# B&R Automation Studio project EFI (part 16)

#### pressureControl.st - Pressure control PID
```iecst
ACTION pressureControl:

	IF inks.parameters.StartUp.xActive THEN
		rMeniscusSp := inks._Internal.Startup.rSetPointMeniscus;
	ELSE
		rMeniscusSp := inks.parSw.NegPump.rSetPointMeniscus;
	END_IF

	xReservoirParamsNeeded := xPressureReservoirStable OR (xReservoirModeActivated AND  mode9); //INKS_STOPPING

	parPidMeniscus:=stPIDParamId(parBar.paramsPidMeniscus);
	xUpdatePidMeniscus:= parPidMeniscusCopy <> parPidMeniscus;
	parPidMeniscusCopy:=parPidMeniscus;
	IF xUpdatePidMeniscus THEN
		iQuantityUpdatePidMeniscus:=iQuantityUpdatePidMeniscus+1;
	END_IF;
	IF xUpdatePidMeniscus OR EDGE(xReservoirParamsNeeded) THEN
		IF NOT xReservoirParamsNeeded THEN
			//Standart values
			stPIDParamToMTPIDParameters(ADR(parBar.paramsPidMeniscus), ADR(pidParMeniscus));
		ELSE
			stPIDParamToMTPIDParameters(ADR(parBar.paramsPidMeniscusReservoir), ADR(pidParMeniscus));
		END_IF
	END_IF;

	parPidPos:=stPIDParamId(parBar.paramsPidPositive);
	xUpdatePidPos:= parPidPosCopy <> parPidPos;
	parPidPosCopy:=parPidPos;
	IF xUpdatePidPos THEN
		iQuantityUpdatePidPos:=iQuantityUpdatePidPos+1;
	END_IF;
	IF xUpdatePidPos OR EDGE(xReservoirParamsNeeded) THEN
		IF NOT xReservoirParamsNeeded THEN
			//Standart values
			stPIDParamToMTPIDParameters(ADR(parBar.paramsPidPositive), ADR(pidParPresPos));
		ELSE
			stPIDParamToMTPIDParameters(ADR(parBar.paramsPidPositiveReservoir), ADR(pidParPresPos));
		END_IF
	END_IF;

	TON_ExecutionDelay(IN:=TRUE, PT:= T#100MS);

	//timer to change the management of the filling pump.
	//Issue 1813: Modification in the change filling control condition, now if the difference between Sp and real meniscus is equal to zero, we change to PID control, too.
	//
	TON_ChangeFillingControl(	IN:=( mode3 AND NOT inks.parameters.Priming.xSystemNeedsPriming AND (rMeniscusError <  LC_MAX_MENISCUS_TO_STARTED)) AND
									( mode3 AND NOT inks.parameters.Priming.xSystemNeedsPriming AND (rMeniscusError >= LC_MIN_MENISCUS_TO_STARTED)) ,
								PT:= T#0.1S);
	IF NOT mode3 THEN
		xGoToStarted := FALSE;
	ELSIF TON_ChangeFillingControl.Q THEN
		xGoToStarted := TRUE;
	END_IF

	IF mode3 AND NOT xPrimingStabilized AND
		( inks.status.PosPump.rDutyCycleFilling > inks.parameters.PosPump.rDCThresholdPriming) AND
		( (rSPfillingPump <> rSP_PressurePos_PID) OR (rMeniscusSp <> rSP_Meniscus_PID) ) THEN

		xPrimingStabilized:=TRUE;
	END_IF

	//Modify the Positive SetPoint during starting
	pressPosAcceleration;

	//**********************************************************************************
	//It changes SP maniscus when is detected differential pressure lower than 20mbars
	//**********************************************************************************
	IF NOT xDrippingOrder THEN

		IF inks.parameters.Priming.xSystemNeedsPriming THEN

			IF mode4 THEN //Inks Started

				// Timer management	for controlling changes in meniscus SP
				TON_ChangeSPstarting(IN:= ( xPrimingStabilized AND (NOT TON_ChangeSPstarting.Q) ), PT:= T#300MS);
				xUpdateSpPriming:= TON_ChangeSPstarting.Q AND inks.status.Temp.rTemp > (rSPtemp-4);

				rPressurePos:= ABS (inks.status.rVacuum1-rSP_PressurePos_PID);
				IF xUpdateSpPriming AND ( rPressurePos < inks.parameters.Priming.rThresholdPressure ) AND (rSPfillingPump <> rSP_PressurePos_PID)  THEN
					// rSPfillingPump is POS PRESSURE SP from GUI

					// rSP_PressurePos_PID current positive pressure sensor
					IF (rSPfillingPump < rSP_PressurePos_PID) THEN
						//Decrease Pos and Meniscus SPs
						rSP_PosPrimStabilizing := rSP_PosPrimStabilizing - 1;
					ELSE
						//Decrease Pos and Meniscus SPs
						rSP_PosPrimStabilizing := rSP_PosPrimStabilizing + 1;
					END_IF
				END_IF

				rPressureMen:= ABS (inks.status.rMeniscus-rSP_Meniscus_PID);
				IF xUpdateSpPriming AND ( rPressureMen < inks.parameters.Priming.rThresholdPressure ) AND  (rMeniscusSp <> rSP_Meniscus_PID) AND (rSPfillingPump = rSP_PressurePos_PID) THEN

					IF (rMeniscusSp < rSP_Meniscus_PID) THEN
						//Decrease Pos and Meniscus SPs
						rSP_NegPrimStabilizing := rSP_NegPrimStabilizing - 1;
					ELSE
						//Decrease Pos and Meniscus SPs
						rSP_NegPrimStabilizing := rSP_NegPrimStabilizing + 1;
					END_IF
				END_IF

				//Update de SetPoints of the PID
				rSP_Meniscus_PID:=rSP_NegPrimStabilizing;
				rSP_PressurePos_PID:=rSP_PosPrimStabilizing;

			END_IF

		ELSE	// THIS IS THE CASE WITHOUT THE PRIMING, THE STANDART BEHAVIOR

			IF xStateReverseFlow THEN

				IF (inks.status.rDeltaPressure <= 20.0) THEN
					rSP_PressurePos_PID := -15.0;
					rSP_Meniscus_PID := 25.0;
				ELSE
					inks.status.startChangeSPInDelta:=TRUE;
				END_IF

			ELSE
				rSP_PressurePos_PID:= rSPfillingPump;
				rSP_Meniscus_PID:=rMeniscusSp;
			END_IF

			// Timer management
			TON_ChangeSPInDelta(IN:=inks.status.startChangeSPInDelta, PT:= SECONDS_TO_TIME(inks.parameters.iTimeChangeSPInRev));
			IF TON_ChangeSPInDelta.Q THEN
				rSP_PressurePos_PID:= rSPfillingPump;
				rSP_Meniscus_PID:=rMeniscusSp;
				inks.status.startChangeSPInDelta:=FALSE;
			END_IF

		END_IF

	ELSE //The ink System has DRIP ORDER

		rSP_Meniscus_PID:=SETPOINT_MENISCUS_DRIP;
		rSP_PressurePos_PID:= -SETPOINT_MENISCUS_DRIP + rSPfillingPump + rMeniscusSp;
		xPrimingStabilized:=FALSE;

	END_IF

	//VACUUM - NEGATIVE - VACUUM - NEGATIVE - VACUUM - NEGATIVE - VACUUM - NEGATIVE - VACUUM - NEGATIVE -
	//VACUUM - NEGATIVE - VACUUM - NEGATIVE - VACUUM - NEGATIVE - VACUUM - NEGATIVE - VACUUM - NEGATIVE -

	//negative pump management.
	iReasonEnableNegPID.0 := mode3;
	iReasonEnableNegPID.1 := mode4;
	iReasonEnableNegPID.2 := mode5;
	iReasonEnableNegPID.3 := mode6;
	iReasonEnableNegPID.4 := mode9;
	xEnableNegPID := iReasonEnableNegPID > 0;

	xHoldMeniscus := (inks.status.iDirection = INKSDIR_REVERSE AND NOT TON_StabSolPid1Neg.Q) OR
					(	NOT TON_StabSolPid2Neg.Q AND
					mode4 AND //INKS_STARTED
					xStateReverseFlow);

	//**********************************************************************************
	// PID PID PID PID PID PID PID PID PID PID PID PID PID PID PID PID PID PID PID PID
	//**********************************************************************************
	fb_PID_Pres(Enable:=xEnableNegPID AND TON_ExecutionDelay.Q,
						PIDParameters:=pidParMeniscus,
						HoldOut:= xHoldMeniscus,
						MinOut:=0.0,
						MaxOut:=100.0,
						Update:= xUpdatePidMeniscus,
						SetValue:=rSP_Meniscus_PID,
						ActValue:=rMeniscusPV
						);
	rOrderBNegative:=fb_PID_Pres.Out;

	//POSITIVE - POSITIVE - POSITIVE - POSITIVE - POSITIVE - POSITIVE - POSITIVE - POSITIVE - POSITIVE - POSITIVE -
	//POSITIVE - POSITIVE - POSITIVE - POSITIVE - POSITIVE - POSITIVE - POSITIVE - POSITIVE - POSITIVE - POSITIVE -

	//filling pump management.
	iReasonEnablePosPID.0 := mode3 AND inks.parameters.Priming.xSystemNeedsPriming;
	iReasonEnablePosPID.1 := mode4;
	iReasonEnablePosPID.2 := mode5;
	iReasonEnablePosPID.3 := mode6;
	iReasonEnablePosPID.4 := mode9;
	xEnablePosPID := iReasonEnablePosPID > 0;

	xHoldPos:= (inks.status.iDirection = INKSDIR_REVERSE AND NOT TON_StabSolPid1Pos.Q) OR
				(NOT TON_StabSolPid2Pos.Q AND
				mode4 AND //INKS_STARTED
				xStateReverseFlow	);

	//**********************************************************************************
	// PID PID PID PID PID PID PID PID PID PID PID PID PID PID PID PID PID PID PID PID
	//**********************************************************************************
	fb_PID_PresFilling(Enable:=xEnablePosPID AND TON_ExecutionDelay.Q,
						PIDParameters:=pidParPresPos,
						HoldOut:= xHoldPos,
						MinOut:=0.0,
						MaxOut:=100.0,
						Update:= xUpdatePidPos,
						SetValue:=rSP_PressurePos_PID,
						ActValue:=rPressureCollectorPos1
						);
	rOrderBPositive:=fb_PID_PresFilling.Out;

	//Define the pump outputs depending on the state

	IF mode3 THEN
		IF inks.parameters.Priming.xSystemNeedsPriming THEN
			rSP_Meniscus_PID	:= inks.parameters.NegPump.rSetPointPrimingStarting;
			rSP_PressurePos_PID	:= inks.parameters.PosPump.rSetPointPrimingStarting;
			inks.status.PosPump.rDutyCycleFilling:=rOrderBPositive;

			//Prepare the initial value for Stabilization stage
			rSP_PosPrimStabilizing:=inks.parameters.PosPump.rSetPointPrimingStarting;
			rSP_NegPrimStabilizing:=inks.parameters.NegPump.rSetPointPrimingStarting;
		ELSE
			rSetPointFillingPump:=parBar.rSPfillingPumpStarting;
			inks.status.PosPump.rDutyCycleFilling:=rOrderBPositiveStart;
		END_IF
		inks.status.NegPump.rDutyCycleNegative:=rOrderBNegative;
	END_IF

	IF NOT mode10 AND (mode4 OR mode5 OR mode6) THEN
		inks.status.PosPump.rDutyCycleFilling:=rOrderBPositive;
		inks.status.NegPump.rDutyCycleNegative:=rOrderBNegative;
	END_IF

	IF mode13 THEN
		inks.status.NegPump.rDutyCycleNegative:=inks.parameters.NegPump.rDCPriming;
		inks.status.PosPump.rDutyCycleFilling:=inks.parameters.PosPump.rDCPriming;
	END_IF

	IF mode10 THEN //InksManifoldCleaning
		inks.status.PosPump.rDutyCycleFilling:=inks.parSw.PosPump.rSetPointManual;
		inks.status.NegPump.rDutyCycleNegative:=inks.parSw.NegPump.rSetPointManual;
	END_IF

	//Sanity checks
	IF mode1 THEN //Inks Stopped
		inks.status.PosPump.rDutyCycleFilling:=0;
		inks.status.NegPump.rDutyCycleNegative:=0;
		xPrimingStabilized:=FALSE;
	END_IF

END_ACTION
```

#### conversionsPost.st - Posconversions
```iecst
ACTION conversionsPost:

	IF  inks.status.xInksRunning THEN

		//Negative Pump
		IF inks.status.NegPump.rDutyCycleNegative=0.0 THEN
			inks.signals.out.iDutyCycleNegative:=0;
		ELSE
			rVoltageNegPump:= (inks.status.NegPump.rDutyCycleNegative * rSlopePumpNeg) + rLowPumpLimitNeg;
			inks.signals.out.iDutyCycleNegative:=REAL_TO_INT(rVoltageNegPump * 32766 / 10); //10V correspond to 32766
		END_IF;

		//Positive Pump
		IF inks.status.PosPump.rDutyCycleFilling=0.0 THEN
			inks.signals.out.iDutyCycleFilling:=0;
		ELSE
			rVoltagePosPump:= (inks.status.PosPump.rDutyCycleFilling * rSlopePumpPos) + rLowPumpLimitPos;
			inks.signals.out.iDutyCycleFilling:=REAL_TO_INT(rVoltagePosPump * 32766 / 10); //10V correspond to 32766
		END_IF;

	ELSE
		inks.signals.out.iDutyCycleNegative:=0;
		inks.signals.out.iDutyCycleFilling:=0;

	END_IF;

	///vars to show in GUI
	inks.status.Tank.iDipositLevel:=REAL_TO_INT(rTankLevelPercent);
	inks.status.tiDriptime:=inks.parSw.tiDripTime;
	inks.status.PosPump.rSetPointPos:=rSP_PressurePos_PID;

	// Duty cycle Heater Tank in Percentage
	inks.status.Temp.rDutyCycleTempPowerRedTank:= inks.status.Temp.rDutyCycleTempTank;   //TOREVIEW: It doesn't seems to be OK (JMH)

END_ACTION
```

#### alarms.st - Alarms
```iecst
ACTION alarms:
	//Ink level alarm
	inks.Al.xAlrTankDigitalSensorsError := NOT inks.status.xActTestMode AND NOT inks.status.Tank.xMinLevel AND inks.status.Tank.xMaxLevel;

	//Temperature and Vacuum probe alarms
	TON_Reset(IN:= NOT xIAmInReverse AND inks.status.xInksRunning, PT:= T#1S);
	t_reset := TON_Reset.Q;

	//Silvia: added an equal symbol in the comparison, because it's impossible to have more than 150mbar.
	TON_AlrVacuum1.IN	:=	t_reset AND (rPressureCollectorPos1 >= rVacuumSensorMax) AND (inks.signals.out.iDutyCycleNegative<>0);
	TON_AlrVacuum1.PT	:=	T#1S; //T#2S; //SUSTPLATF-266
	TON_AlrVacuum1();

	IF TON_AlrVacuum1.Q THEN
		inks.Al.xAlrVacuum1 := TRUE;
	END_IF

	TON_AlrVacuum2.IN	:=	t_reset AND (rPressureCollectorPos2 >= rVacuumSensorMax) AND (inks.signals.out.iDutyCycleFilling<>0);
	TON_AlrVacuum2.PT	:=	T#1S; //T#2S; //SUSTPLATF-266
	TON_AlrVacuum2();

	IF TON_AlrVacuum2.Q THEN
		inks.Al.xAlrVacuum2 := TRUE;
	END_IF

	// Alarm Error in Vacuum gauge means that analog input status is lower than -8000
	TON_DelayVacuum1Gauge.IN	:=	inks.signals.in.xVacuum1SensorError;
	TON_DelayVacuum1Gauge.PT	:=	T#2S;
	TON_DelayVacuum1Gauge();

	IF TON_DelayVacuum1Gauge.Q THEN
		inks.Al.xAlrVacuumSensor1 := TRUE;
	END_IF

	// Alarm Error in Vacuum gauge means that analog input status is lower than -8000
	TON_DelayVacuum2Gauge.IN	:=	inks.signals.in.xVacuum2SensorError;
	TON_DelayVacuum2Gauge.PT	:=	T#2S;
	TON_DelayVacuum2Gauge();

	IF TON_DelayVacuum2Gauge.Q THEN
		inks.Al.xAlrVacuumSensor2 := TRUE;
	END_IF

	TON_AlrVacuumDiff(IN:=t_reset AND ABS(inks.status.rMeniscus-rMeniscusSp) > inks.parSw.NegPump.rLimitMeniscusDiffWarning AND
					NOT inks.Al.xAlrVacuum1 AND	NOT inks.Al.xAlrVacuum2 AND	NOT inks.commands.xErrorRst,
					PT:= T#1S);

	TON_AlrVacuumDiff2(	IN:=mode4 AND ABS(inks.status.rMeniscus-rMeniscusSp) < inks.parSw.NegPump.rLimitMeniscusDiffWarning,
						PT:= T#5S);

	IF TON_AlrVacuumDiff2.Q OR NOT inks.status.xInksRunning THEN
		inks.Al.xAlrDiffVacuum := FALSE;
	// xOrderOnReverseCapped when is cleaning while 50 secs, from start reverse to be finished
	ELSIF TON_AlrVacuumDiff.Q AND NOT xIgnoreAlarmsInCleaning AND NOT inks.status.Reverse.xOnReverseAuto THEN
		inks.Al.xAlrDiffVacuum := TRUE;
	END_IF

	//Temperature alarms management

	//Alarm in the Manifold temperature gauge. (Out of range)
	TON_AlrIncoherTempHeat.IN	:=	t_reset AND ( inks.status.Temp.rTemp < 0.0 OR inks.status.Temp.rTemp > 100.0 );
	TON_AlrIncoherTempHeat.PT	:=	T#2S;
	TON_AlrIncoherTempHeat();

	IF TON_AlrIncoherTempHeat.Q THEN
		inks.Al.xAlrIncoherTempHeat := TRUE;
	END_IF

	//Alarm in Bar Heater temperature gauge. (Out of range)
	TON_AlrTempHeaterMax.IN	:=	(inks.status.Temp.rTemp > 80.0);
	TON_AlrTempHeaterMax.PT	:=	T#2S;
	TON_AlrTempHeaterMax();

	IF TON_AlrTempHeaterMax.Q THEN
		inks.Al.xAlrHeaterReachsMaxTemp := TRUE;
	END_IF

	//////////////////////////////////////////////////////////////////////////////////////////////////////////////////////
	//Alarm of temperature gauge broken temperature gauge in collector. Error detected by the plc
	// COLLECTOR
	// Alarm Error in Vacuum gauge means that analog input status is lower than -8000
	//////////////////////////////////////////////////////////////////////////////////////////////////////////////////////
	TON_AlrTempGauge.IN	:=	(inks.signals.in.xTempSensorError);
	TON_AlrTempGauge.PT	:=	T#2S;
	TON_AlrTempGauge();

	IF TON_AlrTempGauge.Q THEN
		inks.Al.xAlrTempSensor := TRUE;
	END_IF

	alarmsTankHeater;

	//////////////////////////////////////////////////////////////////////////////////////////////////////////////////////
	// Alarm differential temperature
	//////////////////////////////////////////////////////////////////////////////////////////////////////////////////////

	//WARNING

	TON_AlrDifTemp.IN := ABS(inks.status.Temp.rTemp - rSPtemp) > MAX_DIFFCTRLTEMP_WRNG;
	TON_AlrDifTemp.PT := T#2S;
	TON_AlrDifTemp();

	TON_AlrNotDifTemp.IN :=	ABS(inks.status.Temp.rTemp-rSPtemp) < MAX_DIFFCTRLTEMP_WRNG;
	TON_AlrNotDifTemp.PT :=	T#5S;
	TON_AlrNotDifTemp();

	IF NOT inks.status.xInksRunning OR TON_AlrNotDifTemp.Q THEN
		inks.Al.xAlrDiffInCtrlTemp := FALSE;
	ELSIF TON_AlrDifTemp.Q THEN
		inks.Al.xAlrDiffInCtrlTemp := TRUE;
	END_IF

	//ALARM

	IF NOT inks.status.xInksRunning OR NOT inks.status.xEnabledBarToPrint OR TON_AlrNotDifTempExcessiv.Q THEN
		inks.Al.xAlrDifCtrlTempExcessive := FALSE;
	ELSIF TON_AlrDifTempExcessiv.Q THEN
		inks.Al.xAlrDifCtrlTempExcessive := TRUE;
	END_IF

	TON_AlrDifTempExcessiv.IN := ABS(inks.status.Temp.rTemp - rSPtemp) > MAX_DIFFCTRLTEMPHIGH_ALR;
	TON_AlrDifTempExcessiv.PT := T#20s;
	TON_AlrDifTempExcessiv();

	TON_AlrNotDifTempExcessiv.IN := ABS(inks.status.Temp.rTemp - rSPtemp) < MAX_DIFFCTRLTEMPHIGH_ALR;
	TON_AlrNotDifTempExcessiv.PT := T#20s;
	TON_AlrNotDifTempExcessiv();

	//////////////////////////////////////////////////////////////////////////////////////////////////////////////////////
	// Alarm PLC not heating bar
	//////////////////////////////////////////////////////////////////////////////////////////////////////////////////////
	tonAlrNotHeating.IN := inks.status.xInksRunning AND NOT mode10 AND
						(rSPtemp - inks.status.Temp.rTemp > MAX_DIFFCTRLTEMP_ALR) AND
						NOT inks.signals.out.xOutBarResistance;
	tonAlrNotHeating.PT := T#1m;
	tonAlrNotHeating();
	IF tonAlrNotHeating.Q THEN
		IF NOT inks.Al.xAlrHeaterOutFault THEN
			//Added into the IF to avoid a double register while stopping
			LogNotHeating;
		END_IF
		inks.Al.xAlrHeaterOutFault := TRUE;
	END_IF

	//////////////////////////////////////////////////////////////////////////////////////////////////////////////////////
	//Overpressure alarm management
	//////////////////////////////////////////////////////////////////////////////////////////////////////////////////////
	TON_OverPressureDelay.IN := NOT mode1 AND inks.signals.in.xOverpressure;
	TON_OverPressureDelay.PT := T#100ms;
	TON_OverPressureDelay();

	IF TON_OverPressureDelay.Q THEN
		inks.Al.xAlrOverPressure := TRUE;
	END_IF

	//////////////////////////////////////////////////////////////////////////////////////////////////////////////////////
	//Stop Recirculation because there is not ink inn tank
	//////////////////////////////////////////////////////////////////////////////////////////////////////////////////////
	IF (mode3 OR mode13 OR mode4) AND NOT inks.status.Tank.xMinLevel AND NOT inks.status.xActTestMode THEN
		inks.Al.xAlrStopRecircNoInk:=TRUE;
	ELSIF inks.status.Tank.xMinLevel THEN
		inks.Al.xAlrStopRecircNoInk:=FALSE;
	END_IF

	//////////////////////////////////////////////////////////////////////////////////////////////////////////////////////
	// It is defined in controlMode.str_start_inks(CLK:= inks.ordersSw.xStartInks);
	// RECIRCULATION CANNOT START, INK TANK EMPTY
	//////////////////////////////////////////////////////////////////////////////////////////////////////////////////////
	IF NOT inks.status.xActTestMode AND NOT inks.status.Tank.xMinLevel AND r_start_inks.Q THEN
		inks.Al.xAlrInksRunnig:=TRUE; //To review with Jorge, this alarm is not shared in VarsVersion but exists in PLC2Kernel
	END_IF

	//////////////////////////////////////////////////////////////////////////////////////////////////////////////////////
	// Implemented 09/19/2017
	// Here, an alarm No Recirculation in the Bar is reported when is Ink system is stopped with bar installed
	// RECIRCULATION STOPPED / UNSTABLE INK SYSTEM
		//////////////////////////////////////////////////////////////////////////////////////////////////////////////////////
	inks.Al.xAlrNoRecirculation :=  NOT inks.status.xInksRunning;

	//////////////////////////////////////////////////////////////////////////////////////////////////////////////////////
	//INK SYSTEM STOPED WITH BAR ENABLE TO PRINT
	//////////////////////////////////////////////////////////////////////////////////////////////////////////////////////
	IF NOT inks.status.xInksRunning AND inks.status.xEnabledBarToPrint THEN
		inks.Al.xAlrNoRecircStop := TRUE;
	END_IF

	//////////////////////////////////////////////////////////////////////////////////////////////////////////////////////
	//Alarm to indicate that we don't allow to enter in the  manifold cleaning mode if there is no ink.
		//////////////////////////////////////////////////////////////////////////////////////////////////////////////////////
	IF NOT inks.status.xActTestMode AND NOT inks.status.Tank.xMinLevel AND EDGEPOS(inks.ordersSw.xStartManual) THEN
		inks.Al.xAlrNoInkNoCleanManif := TRUE;
	END_IF

	// rSPfillingPump is POS PRESSURE SP from GUI
	// rSP_PressurePos_PID current positive pressure sensor
	// rMeniscusSp is Meniscus SP from GUI
	// rSP_Meniscus_PID current meniscus pressure
	xOutOfCriticalRange := 	mode4 AND (rSPfillingPump = rSP_PressurePos_PID) AND (rMeniscusSp = rSP_Meniscus_PID) AND
				( rMeniscusPV > inks.parSw.NegPump.rUpperLimMeniscusCritical  OR  rMeniscusPV < inks.parSw.NegPump.rLowerLimMeniscusCritical );

	TON_AlrCriticalMeniscus2.IN:=t_reset AND mode4 AND NOT xIgnoreAlarmsInCleaning AND xOutOfCriticalRange;
	TON_AlrCriticalMeniscus2.PT:=T#5S;
	TON_AlrCriticalMeniscus2();

	IF TON_AlrCriticalMeniscus2.Q THEN
		inks.Al.xAlrBrokenMeniscus := TRUE;
	END_IF

	IF inks.status.xActTestMode THEN
		inks.Al.xAlrLevelSensorError := FALSE;
	ELSIF inks.status.Tank.xMaxLevel AND NOT inks.status.Tank.xMinLevel THEN
		inks.Al.xAlrLevelSensorError := TRUE;
	END_IF

	// It is not a stop alarm just warning
	inks.Al.xAlrTankToFillIn := NOT inks.status.xActTestMode AND NOT inks.status.Tank.xMaxLevel;

	// It has been improved to avoid zero state in the machine when this alarm is activated. Added condition status is different to mode1
	// 22-10-1017: Changed for commissioning SN1 at Marco Polo: It is alarm stop when inkState is different to INKS_STOPPED
	inks.Al.xAlrTankEmpty := NOT inks.status.xActTestMode AND NOT mode1 AND NOT inks.status.Tank.xMinLevel;

	// The ink level is close to Empty. Raising an alarm to allow the Machine or the line to stop production without stopping the inkSystem
	inks.Al.xAlrTankCloseToEmpty := NOT inks.status.xActTestMode AND NOT mode1 AND NOT inks.status.Tank.xCloseToMinLevel;

	TON_TimeAlrDCStarting(IN:=mode3, PT:= T#60S);  //After start, delay 60seconds taking care of this alarm

	xModesAlrDC:=TON_TimeAlrDCStarting.Q OR (mode4 AND NOT xIgnoreAlarmsInCleaning );

	TON_AlrDCDiff.IN:= xModesAlrDC AND ABS(inks.status.PosPump.rDutyCycleFilling - inks.status.NegPump.rDutyCycleNegative) > lc_rDiffBetweenPumpsDCLimit;
	TON_AlrDCDiff.PT:= inks.parameters.parBar.iTimeToActiveDcErrorAlarm;
	TON_AlrDCDiff();

	TON_AlrNegDiff.IN:= xModesAlrDC AND ( (inks.status.NegPump.rDutyCycleNegative>99) OR (inks.status.NegPump.rDutyCycleNegative < 1 ));
	TON_AlrNegDiff.PT:= inks.parameters.parBar.iTimeToActiveDcErrorAlarm;
	TON_AlrNegDiff();

	TON_AlrPosDiff.IN:= xModesAlrDC AND ( (inks.status.PosPump.rDutyCycleFilling>99) OR (inks.status.PosPump.rDutyCycleFilling < 1 ));
	TON_AlrPosDiff.PT:= inks.parameters.parBar.iTimeToActiveDcErrorAlarm;
	TON_AlrPosDiff();

	IF TON_AlrDCDiff.Q OR TON_AlrNegDiff.Q OR TON_AlrPosDiff.Q THEN
		inks.Al.xAlrPumpsDCError := TRUE;
		LogPumpDCError; //Logging the source of the Pump DC Error
	END_IF

	IF inks.signals.in.xKlixonTriggered THEN
		inks.Al.xAlrKlixonTriggered:=TRUE;
	// This ELSE must be reviewed with Dani Moya, added during Cube start up.
	ELSE
		inks.Al.xAlrKlixonTriggered:=FALSE;
	END_IF

	// It allows detection because PsuOk is delayed when is in failure
	TON_StabPsuOk.IN:=(inks.ordersSw.xPowPrintHead AND inks.signals.out.xOutPowPrintHead AND NOT inks.signals.in.xPrintHeadsPsuOK);
	TON_StabPsuOk.PT:=lc_tiTimeStoppingPsu;
	TON_StabPsuOk();

	IF TON_StabPsuOk.Q THEN
		inks.Al.xAlrPrintHeadPsuFailure:=TRUE;
	END_IF

	//DELOREAN-1961: Warning when bar enabled to print and maintenance mode active
	IF inks.status.xActMaintenanceMode AND inks.status.xEnabledBarToPrint THEN
		inks.Al.xAlrMaintenanceModeActive := TRUE;
	END_IF

	// NOZOMITWO-1410 Chiller alarms
	TON_AlrHeaterOFF.IN := inks.status.xInksRunning AND inks.parameters.InksChiller.Status=CHILLER_RUNNING AND inks.signals.out.xHeatingActive AND inks.status.Temp.rDutyCycleTemp = 0 AND (inks.parSw.Temp.rSetPointTemp + 1) < inks.status.Temp.rTemp;
	TON_AlrHeaterOFF.PT := T#120s;
	TON_AlrHeaterOFF();

	inks.Al.xHeaterOff := TON_AlrHeaterOFF.Q;

	// NOZOMITWO-1410 Chiller warnings and NOZOMITWO-2353
	TON_AlrChillerPrintheadsOFF.IN := inks.parameters.PrintheadsChiller.iIndex > 0 AND
									inks.parameters.PrintheadsChiller.Status <> CHILLER_RUNNING AND
									inks.parameters.PrintheadsChiller.Status <> CHILLER_STOPPING AND
									inks.signals.out.xOutPowPrintHead;
	TON_AlrChillerPrintheadsOFF.PT := T#30s;
	TON_AlrChillerPrintheadsOFF();

	IF TON_AlrChillerPrintheadsOFF.Q THEN
		inks.Al.xAlrPrintHeadsChillerStopped := TRUE;
	END_IF

END_ACTION

ACTION alarmsTankHeater:

	IF NOT inks.parSw.Temp.xTankHeaterEnabled THEN
		inks.Al.xAlrTempTankSensor			:= FALSE;
		inks.Al.xAlrHeaterTankReachsMaxTemp	:= FALSE;
		inks.Al.xAlrDiffInCtrlTempTank		:= FALSE;
		inks.Al.xAlrIncoherTempTank			:= FALSE;
		RETURN;
	END_IF

	//////////////////////////////////////////////////////////////////////////////////////////////////////////////////////
	//Alarm temperature gauge broken in heater or temperature gauge broken HEATER TANK. Error detected by the plc.
	// xTempTankSensorError --> It has not I/O mapping. Pending to define in P4	by EEteam
	//HEATER TANK
	//////////////////////////////////////////////////////////////////////////////////////////////////////////////////////

	TON_AlrTempTankTempSensorError.IN	:=	inks.signals.in.xTempTankSensorError;
	TON_AlrTempTankTempSensorError.PT	:=	T#2S;
	TON_AlrTempTankTempSensorError();

	// If not installed bar en It is not an alarm
	IF TON_AlrTempTankTempSensorError.Q THEN
		inks.Al.xAlrTempTankSensor := TRUE;
	END_IF

	//Alarm in Heater Tank temperature gauge. (Out of range)
	TON_AlrTempTankMax.IN	:=	(inks.status.Temp.rTempTank > 70.0);
	TON_AlrTempTankMax.PT	:=	T#2S;
	TON_AlrTempTankMax();

	IF TON_AlrTempTankMax.Q THEN
		inks.Al.xAlrHeaterTankReachsMaxTemp := TRUE;
	END_IF

	//Alarm differential temperature in tank
	TON_AlrDifTempTank.IN	:=	t_reset AND ( ABS(inks.status.Temp.rTempTank - rSPTempTank) > MAX_DIFFCTRLTEMP_WRNG);
	TON_AlrDifTempTank.PT	:=	T#2S;
	TON_AlrDifTempTank();

	TON_AlrDifTempTank2.IN	:=	inks.status.xInksRunning AND (ABS(inks.status.Temp.rTempTank-rSPTempTank) < MAX_DIFFCTRLTEMP_WRNG);
	TON_AlrDifTempTank2.PT	:=	T#5S;
	TON_AlrDifTempTank2();

	IF NOT inks.status.xInksRunning OR TON_AlrDifTempTank2.Q THEN
		inks.Al.xAlrDiffInCtrlTempTank := FALSE;
	ELSIF TON_AlrDifTempTank.Q THEN
		inks.Al.xAlrDiffInCtrlTempTank := TRUE;
	END_IF

	//Alarm in the heater tank temperature gauge. (Out of range)
	TON_AlrIncoherTempTank.IN	:=	t_reset AND ( inks.status.Temp.rTempTank < 0.0 OR inks.status.Temp.rTempTank > 100.0 );
	TON_AlrIncoherTempTank.PT	:=	T#2S;
	TON_AlrIncoherTempTank();

	IF TON_AlrIncoherTempTank.Q THEN
		inks.Al.xAlrIncoherTempTank := TRUE;
	END_IF
END_ACTION

ACTION LogPumpDCError:

	IF inks.status.NegPump.rDutyCycleNegative>99 THEN
		stEventLogNeg.Source := ELOG_TYPE_BAR;
		stEventLogNeg.Severity:= ELOG_SEVERITY_ERROR;
		stEventLogNeg.Facility:= gIndexInks;
		stEventLogNeg.ErrorCode:=0;
		stEventLogNeg.Text := 'Negative Pump in Max Value. Bar ';
		brsftoa(gIndexInks, ADR(strAux));
		brsstrcat(ADR(stEventLogNeg.Text), ADR(strAux));
		gEventLogLoader(EventData := ADR(stEventLogNeg));
	END_IF
	IF inks.status.NegPump.rDutyCycleNegative<1 THEN
		stEventLogNeg.Source := ELOG_TYPE_BAR;
		stEventLogNeg.Severity:= ELOG_SEVERITY_ERROR;
		stEventLogNeg.Facility:= gIndexInks;
		stEventLogNeg.ErrorCode:=0;
		stEventLogNeg.Text := 'Negative Pump in Min Value. Bar ';
		brsftoa(gIndexInks, ADR(strAux));
		brsstrcat(ADR(stEventLogNeg.Text), ADR(strAux));
		gEventLogLoader(EventData := ADR(stEventLogNeg));
	END_IF
	IF inks.status.PosPump.rDutyCycleFilling>99 THEN
		stEventLogPos.Source := ELOG_TYPE_BAR;
		stEventLogPos.Severity:= ELOG_SEVERITY_ERROR;
		stEventLogPos.Facility:= gIndexInks;
		stEventLogPos.ErrorCode:=0;
		stEventLogPos.Text := 'Filling Pump in Max Value. Bar ';
		brsftoa(gIndexInks, ADR(strAux));
		brsstrcat(ADR(stEventLogPos.Text), ADR(strAux));
		gEventLogLoader(EventData := ADR(stEventLogPos));
	END_IF
	IF inks.status.PosPump.rDutyCycleFilling<1 THEN
		stEventLogPos.Source := ELOG_TYPE_BAR;
		stEventLogPos.Severity:= ELOG_SEVERITY_ERROR;
		stEventLogPos.Facility:= gIndexInks;
		stEventLogPos.ErrorCode:=0;
		stEventLogPos.Text := 'Filling Pump in Min Value. Bar ';
		brsftoa(gIndexInks, ADR(strAux));
		brsstrcat(ADR(stEventLogPos.Text), ADR(strAux));
		gEventLogLoader(EventData := ADR(stEventLogPos));
	END_IF

END_ACTION

ACTION LogNotHeating:

	stEventLog.Source := ELOG_TYPE_BAR;
	stEventLog.Severity:= ELOG_SEVERITY_ERROR;
	stEventLog.Facility:= gIndexInks;
	stEventLog.ErrorCode:=0;
	stEventLog.Text := 'Not Heating Error. Bar ';
	brsftoa(gIndexInks, ADR(strAux));
	brsstrcat(ADR(stEventLog.Text), ADR(strAux));
	gEventLogLoader(EventData := ADR(stEventLog));

END_ACTION
```

#### EventLog.st
```iecst
ACTION LogStopAlarm:

	stStopAlarmsLog.Source := ELOG_TYPE_BAR;
	stStopAlarmsLog.Severity:= ELOG_SEVERITY_INFO;
	stStopAlarmsLog.Facility:= 0;
	stStopAlarmsLog.ErrorCode:=0;

	stStopAlarmsLog.Text := 'Inks.LogStopAlarm';

	IF iReasonStop.0 THEN stStopAlarmsLog.Text := 'iReasonCritical > 0';
	ELSIF iReasonStop.1 THEN stStopAlarmsLog.Text := 'inks.Al.xAlrHeaterOutFault';
	ELSIF iReasonStop.2 THEN stStopAlarmsLog.Text := 'inks.Al.xAlrPrintHeadPsuFailure';
	ELSIF iReasonStop.3 THEN stStopAlarmsLog.Text := 'inks.Al.xAlrDifCtrlTempExcessive';
	ELSIF iReasonStop.4 THEN stStopAlarmsLog.Text := 'NOT inks.ordersSw.xStartInks';
	ELSIF iReasonStop.5 THEN stStopAlarmsLog.Text := 'inks.parSw.Config.iInkType = 0';
	ELSIF iReasonStop.6 THEN stStopAlarmsLog.Text := 'inks.parSw.Config.iPrintHeadType = 0';
	ELSIF iReasonStop.7 THEN stStopAlarmsLog.Text := 'inks.Al.xAlrNoRecircStop';
	ELSIF iReasonStop.8 THEN stStopAlarmsLog.Text := 'inks.Al.xAlrTankCloseToEmpty';
	ELSIF iReasonStop.9 THEN stStopAlarmsLog.Text := 'inks.Al.xAlrPrintHeadsChillerStopped';
	END_IF

	gEventLogLoader(EventData := ADR(stStopAlarmsLog));

END_ACTION

ACTION LogCriticalAlarm:

	stEventLogCritical.Source := ELOG_TYPE_BAR;
	stEventLogCritical.Severity:= ELOG_SEVERITY_ERROR;
	stEventLogCritical.Facility:= gIndexInks;
	stEventLogCritical.ErrorCode:=0;

	stEventLogCritical.Text := 'Inks.LogCriticalAlarm';

	IF 		iReasonCritical.0 THEN stEventLogCritical.Text := 'Bar. xAlrTankEmpty';
	ELSIF 	iReasonCritical.1 THEN stEventLogCritical.Text := 'Bar. xAlrStopRecircNoInk';
	ELSIF 	iReasonCritical.2 THEN stEventLogCritical.Text := 'Bar. xAlrTemp';
	ELSIF 	iReasonCritical.3 THEN stEventLogCritical.Text := 'Bar. xAlrVacuum1';
	ELSIF 	iReasonCritical.4 THEN stEventLogCritical.Text := 'Bar. xAlrVacuum2';
	ELSIF 	iReasonCritical.5 THEN stEventLogCritical.Text := 'Bar. xAlrVacuumSensor1';
	ELSIF 	iReasonCritical.6 THEN stEventLogCritical.Text := 'Bar. xAlrVacuumSensor2';
	ELSIF 	iReasonCritical.7 THEN stEventLogCritical.Text := 'Bar. xAlrTempSensor';
	ELSIF 	iReasonCritical.8 THEN stEventLogCritical.Text := 'Bar. xAlrBrokenMeniscus';
	ELSIF 	iReasonCritical.9 THEN stEventLogCritical.Text := 'Bar. xAlrOverPressure';
	ELSIF 	iReasonCritical.10 THEN stEventLogCritical.Text := 'Bar. xAlrLevelSensorError';
	ELSIF 	iReasonCritical.11 THEN stEventLogCritical.Text := 'Bar. xAlrTankDigitalSensorsError';
	ELSIF 	iReasonCritical.12 THEN stEventLogCritical.Text := 'Bar. xAlrPumpsDCError';
	ELSIF 	iReasonCritical.13 THEN //stEventLog.Text := 'Bar. xAlrTemp';
	ELSIF 	iReasonCritical.14 THEN //stEventLog.Text := 'Bar. xAlrTemp';
	ELSIF 	iReasonCritical.15 THEN //stEventLog.Text := 'Bar. xAlrTemp';
	END_IF

	gEventLogLoader(EventData := ADR(stEventLogCritical));

END_ACTION
```

#### inkStateValue.st - Ink values
```iecst
(* TODO: Add your comment here *)
FUNCTION inkStateValue

	CASE inkState OF
		INKS_STOPPED:
			inkStateValue:= 1;

		INKS_STARTING:
			inkStateValue:= 3;

		INKS_STARTED:
			inkStateValue:= 4;

		INKS_MANUAL_REVERSEFLOW:
			inkStateValue:= 5;

		INKS_AUTO_REVERSEFLOW:
			inkStateValue:= 6;

		INKS_STOPPING:
			inkStateValue:= 9;

		INKS_RUNNING_MANUAL:
			inkStateValue:= 10;

		ELSE
			inkStateValue:= 255;

	END_CASE;

END_FUNCTION

(*
INKS_STOPPED					1	 	 	 	252
INKS_DRAINAGE				2	 	 	 	253
INKS_STARTING				3	 	 	 	254
INKS_STARTED					4	 	 	 	255
INKS_MANUAL_REVERSEFLOW		5	 	 	 	256
INKS_AUTO_REVERSEFLOW	6	 	 	 	257
INKS_STOPPING				9	 	 	 	260
INKS_RUNNING_MANUAL		10	 	 	 	261
INKS_UNDEFINED				255	 	 	 	262
*)
```

#### timeToStartPWM.st - Limit power in psu heater
```iecst
(* TODO: Add your comment here *)
FUNCTION timeToStartPWM

//	iItemNumber	INT	FALSE	VAR_INPUT
//	iTotalItems	INT	FALSE	VAR_INPUT
//	iTaskCycle	UINT	FALSE	VAR_INPUT
//	iMsInCycle	UINT		VAR_IN_OUT

	iMsInCycle := UDINT_TO_UINT(TIME_TO_UDINT(clock_ms()) MOD (REAL_TO_UDINT(lc_rCyclePwm) * 1000) );

	IF iTotalItems = 1 THEN
		timeToStartPWM := TRUE;
	ELSIF iTotalItems = 0 THEN
		timeToStartPWM := FALSE;
	ELSE
		timeToStartPWM := 	iMsInCycle >= REAL_TO_UINT(INT_TO_REAL(iItemNumber) * (lc_rCyclePwm * 1000 / INT_TO_REAL(iTotalItems)))  AND
							iMsInCycle<= REAL_TO_UINT(INT_TO_REAL(iItemNumber) * (lc_rCyclePwm * 1000 / INT_TO_REAL(iTotalItems)) + UINT_TO_REAL(iTaskCycle));
	END_IF

END_FUNCTION
```

### InksSim.var
```iecst
VAR
	iInksSimIndex : USINT;
END_VAR
```

- Program Logical/ExtPack/InksCtrl/InksSim/InksSim_v1/InitInksSim (IEC) (no source held here)

### InkSim.var
```iecst
VAR
	simPresPos : SimAnalogProcess; (*Function block to simulate the positive pressure of the inks*)
	simPresNeg : SimAnalogProcess; (*Function block to simulate the meniscus of the inks*)
	simTemp : SimAnalogProcess; (*Function block to simulate the temperature of the inks*)
	xStarted : BOOL;
	Inks : REFERENCE TO stInks;
	tonNotHeating : TON;
	SimInks : REFERENCE TO SimInk_typ;
END_VAR
```

### Program Logical/ExtPack/SimpleBlockCtrl/SimpleBlockCtrl_v1/SimpleBlockCtrl (IEC) - Block program

#### BlockAlarms.st - Block alarms
```iecst
ACTION BlockAlarms:

	// Alarm: Reference incoherence  (NEW: Add To Software)
	T_DelayAlarmRef.IN:=Block.In.xReferenceDI <> AxisBK.Status.DigitalInputs.RefSwitch;
	T_DelayAlarmRef.PT:=T#1000ms;
	T_DelayAlarmRef();

	Block.Al.xAlrReferenceIncoherence:= T_DelayAlarmRef.Q;

	// Alarm: Drive protection
	IF NOT Block.In.xDriveProtectionOK THEN
		Block.Al.xAlrDriveProtection:= TRUE;
	END_IF

	// Alarm: Temp Vertical Motor
	IF AxisBK.Status.ActTempMot > (AxisBK.Status.MaxTempMotor - 5.0) THEN
		IF AxisBK.Status.MaxTempMotor > 0 THEN Block.Al.xBarMotorTemp := TRUE; END_IF
	ELSIF AxisBK.Status.ActTempMot < (AxisBK.Status.MaxTempMotor - 7.0) THEN
		Block.Al.xBarMotorTemp := FALSE;
	END_IF

	// Alarm: Temp Vertical Driver
	IF AxisBK.Status.ActTempDrv > (AxisBK.Status.MaxTempDrv - 5.0) THEN
		IF AxisBK.Status.MaxTempDrv > 0 THEN Block.Al.xBarDriverTemp := TRUE; END_IF
	ELSIF AxisBK.Status.ActTempDrv < (AxisBK.Status.MaxTempDrv - 7.0) THEN
		Block.Al.xBarDriverTemp := FALSE;
	END_IF

	//Not homed bar motor.
	Block.Al.xAlrBarMtrNoRef:= NOT Block.Status.Motor.xBarsHomed;

	//DRIVE ALARMS
	//Comms error in bar motor
	// Pass codes to ennum type 32189
	Block.Al.xAlrComBarMtr:= (AxisBK.Status.ErrorID= 29265)OR (AxisBK.Status.ErrorID= 32189);

	// Alarm: Any drive Alarm
	//Silvia: if there machine is in zero, we don't activate the alarms.
	TON_DelayAnyDriveAlarm.IN:= AxisBK.Status.ErrorID<>0 AND NOT Block.AlSummary.xAlrSafetySystemGeneral AND NOT Block.commands.Mode.xZero AND NOT Block.commands.AutoMode.xBypass;
	TON_DelayAnyDriveAlarm.PT:=t#200ms;
	TON_DelayAnyDriveAlarm();
	Block.Al.xAnyDriveAlarm:= TON_DelayAnyDriveAlarm.Q;

	// Alarm: Power Error
	//Silvia: this alarm was not well assotiated.
	Block.Al.xAlBarMotorPowerOff:= NOT Block.In.xDriveProtectionOK;//AxisBK.Status.ErrorID=5012;

	//Warning: Check Homing Sensor Broken
	IF Block.Al.xAnyDriveAlarm AND (Block.Status.PositionState = BLOCKP_HOMING_BAR) THEN
		Block.Al.xAlrCheckHomingSensor:=TRUE;
	END_IF

	//Maxium bars lifting alarm
	IF rMotorCurrentPos >= Block.parameters.Motor.rSafePosition THEN
		Block.Al.xAlrBlockReachedMaxPosition := TRUE;
	END_IF

	TNotPrinterZero.IN:=NOT Block.commands.Mode.xZero;
	TNotPrinterZero.PT:=T#500ms;
	TNotPrinterZero();

	//########################## ALARMS SUMMARY ########################################
	AlarmsSummary;

END_ACTION
```

#### BlockStatePos.st
```iecst
ACTION BlockStatePos:

	xBlockPosChange := BlockPositionPrevious <> Block.Status.PositionState;
	BlockPositionPrevious := Block.Status.PositionState;

	CASE Block.Status.PositionState OF
		BLOCKP_UNDEFINED:
			ResetKnownPositions;

		BLOCKP_HOMING_BAR:

			//Aborting Block Motor homing process
			iCancelHomingBar.2 := Block.AlSummary.xAlarmCritical;
			iCancelHomingBar.3 := Block.commands.Mode.xZero;
			iCancelHomingBar.4 := NOT Block.commands.xBarHomeOrder;
			IF iCancelHomingBar > 0 THEN
				ResetHomingBar;
				Block.Status.PositionState := BLOCKP_UNDEFINED;
			END_IF

			HomingBar;
			IF Block.Status.Motor.xBarsHomed THEN
				Block.Status.PositionState := BLOCKP_UNDEFINED;
			END_IF

		BLOCKP_IN_CAP:

		BLOCKP_IN_PRINT:

			//Send and adjustment in position if needed
			IF ABS(rMotorCurrentPos-rCalcPosDesPrint)>0.01 AND rMotorAbsPosDesired <> rCalcPosDesPrint THEN

				rMotorAbsPosDesired:= rCalcPosDesPrint;
				xMotorAbsMovOrder:= TRUE;

			END_IF

			Block.Status.Position.xReadyToPrint := rMotorCurrentPos = rCalcPosDesPrint;

		BLOCKP_GOING_TO_CAP:
			GoingToCap;
			IF xInCap THEN
				Block.Status.PositionState := BLOCKP_IN_CAP;
			END_IF

		BLOCKP_GOING_TO_PRINT:
			GoingToPrint;
			IF xInPrint THEN
				Block.Status.PositionState := BLOCKP_IN_PRINT;
			END_IF

	END_CASE

END_ACTION
```

#### ManualLogic.st
```iecst
ACTION ManualMovements:

	IF Block.commands.xBarHomeOrder OR Block.commands.xReset THEN
		RETURN;
	END_IF

	// Excessive Motor block activated
	TON_excessiveBlockActivated.IN:= Block.commands.Mode.xManual AND
									(AxisBK.Command.Jog.ContinuousPos OR
									AxisBK.Command.Jog.ContinuousNeg OR
									Block.commands.Manual.xManBarsUp OR
									Block.commands.Manual.xManBarsDown );
	TON_excessiveBlockActivated.PT:= T#500MS;
	TON_excessiveBlockActivated();
	xStoppedByExcessiveTimeActive:=TON_excessiveBlockActivated.Q;

	IF xStoppedByExcessiveTimeActive OR EDGEPOS(xChangeMotorSpeedUp) OR EDGEPOS(xChangeMotorSpeedDown) THEN
		Block.commands.Manual.xManBarsUp := FALSE;
		Block.commands.Manual.xManBarsDown := FALSE;
	END_IF

	// Enable Up and Down movements if AnyBarEnabled
	IF NOT xStoppedByExcessiveTimeActive THEN

		Block.Status.Motor.xEnableUp:= 	(Block.commands.Mode.xManual AND NOT Block.Status.Motor.xBarsHomed) OR //Silvia: conditions for moving when the motor is not homed (issue 1283).
										(Block.Status.Motor.xBarsHomed AND (rMotorCurrentPos<=Block.parameters.Motor.rSafePosition)); // Lower than max is allowing to go up

		Block.Status.Motor.xEnableDown:= (Block.Status.Motor.xBarsHomed ) OR // <357 mm position max on venturi
										( Block.Status.Motor.xBarsHomed ) OR // 335.5 mm position max on venturi
										(Block.Status.Motor.xBarsHomed AND rMotorCurrentPos> Block.parameters.Motor.rMinSafePosition) OR
										(NOT Block.Status.Motor.xBarsHomed AND (NOT Block.Al.xAlrReferenceIncoherence AND Block.In.xReferenceDI)); //Silvia: issue 1283: we cannot move bars with the sensor broken.
	ELSE
		Block.Status.Motor.xEnableUp:=FALSE;
		Block.Status.Motor.xEnableDown:=FALSE;
	END_IF;

	////////////////
	// Block Motor
	////////////////

	// Moving up
	AxisBK.Command.Jog.ContinuousPos:= Block.Status.Motor.xEnableUp AND Block.commands.Manual.xManBarsUp AND NOT Block.commands.Manual.xManBarsDown;

	// Moving down
	AxisBK.Command.Jog.ContinuousNeg:= Block.Status.Motor.xEnableDown AND Block.commands.Manual.xManBarsDown AND NOT Block.commands.Manual.xManBarsUp;

	// Change vel.
	ManualSpeedControl;

	//Go to Undefined if any movement is raised during Manual
	iReasonMovingMan.0 := AxisBK.Command.Jog.ContinuousPos;
	iReasonMovingMan.1 := AxisBK.Command.Jog.ContinuousNeg;
	IF iReasonMovingMan >0 THEN
		Block.Status.PositionState := BLOCKP_UNDEFINED;
	END_IF

	//First Home direct to enable movement of the drive
	IF 	NOT AxisBK.Status.HomeOK AND NOT Block.Status.Motor.xBarsHoming THEN
		//AxisBK.Parameter.HomePosition:=AxisBK.Status.ActPosition;
		AxisBK.Command.HomeDirect:=TRUE;
	END_IF

END_ACTION

ACTION HomingBar:

	IF xBlockPosChange THEN
		AxisBK.Command.QuickStop:=FALSE;				// Reset state QuickStop
		nState := 150;
	END_IF

	CASE nState OF

		(*----------------------------------- BAR HOMING ----------------------------------------------------------*)
		(*----------------------------------- BAR HOMING ----------------------------------------------------------*)
		(*----------------------------------- BAR HOMING ----------------------------------------------------------*)

		150:
			iLastState:=nState;
			Block.Status.Motor.xBarsHomed:= FALSE;
			AxisBK.Status.HomeOK := FALSE;
			xMotorHomeOrder:= TRUE;
			nState:=nState+1;

		151:
			iLastState:=nState;
			IF AxisBK.Status.HomeOK THEN
				xMotorHomeOrder:= FALSE;
				Block.commands.xBarHomeOrder:=FALSE;
				Block.Status.Motor.xBarsHomed:= TRUE;
				nState:= 0;
			END_IF

	END_CASE

END_ACTION

ACTION ManualSpeedControl:

	IF NOT Block.Status.Motor.xBarsHomed THEN
		xChangeMotorSpeedUp		:= FALSE;
		xChangeMotorSpeedDown	:= FALSE;
		RETURN;
	END_IF

	IF AxisBK.Command.Jog.ContinuousNeg THEN //DOWN

		xChangeMotorSpeedUp := FALSE;

		IF rMotorCurrentPos <= Block.parameters.Motor.rMinSafePosition + Block.parameters.Motor.rReduceSpeedDistance THEN

			xChangeMotorSpeedDown := TRUE;

		END_IF

	ELSIF AxisBK.Command.Jog.ContinuousPos THEN //UP

		xChangeMotorSpeedDown := FALSE;

		IF rMotorCurrentPos >= Block.parameters.Motor.rSafePosition - Block.parameters.Motor.rReduceSpeedDistance THEN

			xChangeMotorSpeedUp := TRUE;

		END_IF

	ELSIF NOT ((rMotorCurrentPos <= Block.parameters.Motor.rMinThicknessMedia + Block.parameters.Motor.rReduceSpeedDistance) OR
		(rMotorCurrentPos >= Block.parameters.Motor.rSafePosition - Block.parameters.Motor.rReduceSpeedDistance)) THEN

		xChangeMotorSpeedUp		:= FALSE;
		xChangeMotorSpeedDown	:= FALSE;

	END_IF

END_ACTION
```

#### ResetCommands.st
```iecst
ACTION ResetHomingBar:

	xMotorHomeOrder := FALSE;
	Block.commands.xBarHomeOrder:=FALSE;
	iTimesStopMovWhileHoming := iTimesStopMovWhileHoming + 1;

	StopBar;

END_ACTION

ACTION StopBar:

	AxisBK.Command.Jog.ContinuousNeg:= FALSE;
	AxisBK.Command.Jog.ContinuousPos:= FALSE;
	IF AxisBK.Status.PLCopenState.ContinuousMotion OR AxisBK.Status.PLCopenState.DiscreteMotion THEN
		AxisBK.Command.Move.Halt:=TRUE;
	ELSIF AxisBK.Status.PLCopenState.Homing THEN
		AxisBK.Command.QuickStop:=TRUE;
	ELSIF NOT AxisBK.Status.PLCopenState.Homing THEN
		AxisBK.Command.QuickStop:=FALSE;
	END_IF

END_ACTION

ACTION ResetEdgeCommands:

	Block.commands.xToCapLab := FALSE;
	Block.commands.xToPrintLab := FALSE;

END_ACTION
```

#### InputParamsMotors.st - Send params to icla and block axis
```iecst
ACTION InputParamsMotors:

	//MOTOR   MOTOR   MOTOR   MOTOR   MOTOR   MOTOR   MOTOR   MOTOR   MOTOR   MOTOR
	//MOTOR   MOTOR   MOTOR   MOTOR   MOTOR   MOTOR   MOTOR   MOTOR   MOTOR   MOTOR
	//MOTOR   MOTOR   MOTOR   MOTOR   MOTOR   MOTOR   MOTOR   MOTOR   MOTOR   MOTOR

	MotorDriveUnit.TransmissionData:=Block.parameters.Motor.DriveUnit;

	// PowerOn Command
	AxisBK.Command.Power:= 	NOT Block.Al.xAlrSafetySystemInBlock AND
							AxisBK.Status.ControllerReady AND
							AxisBK.Status.InitDone;

	// In (mm *10)
	IF AxisBK.Status.HomeOK THEN MotorDriveUnit.pulsesDevice := AxisBK.Status.ActPosition; END_IF //TODO: Remove the HomeOK condition. Now to avoid the NotANumer error
	MotorDriveUnit.Calculation := CALC_POS_MM;
	MotorDriveUnit();
	rMotorCurrentPos:=MotorDriveUnit.PositionDevice;
	Block.Status.rMotorPosition:=rMotorCurrentPos; //Use internal var to assign it

	//Log the Position after to be in position
	IF EDGEPOS(AxisBK.Status.InPosition) THEN
		LogVertInPosition;
	END_IF

	// Position for absolute movement order	// In (mm *10)
	// Move Absolute
	MotorDriveUnit.PositionDesired := rMotorAbsPosDesired;
	MotorDriveUnit.Calculation := CALC_POS_PULSES;
	MotorDriveUnit();
	AxisBK.Parameter.Position:= MotorDriveUnit.pulsesPositionDesired;

	// Auto Acceleration, Velocity Movements
	//AxisBK.Parameter.Acceleration:=	250000;
	MotorDriveUnit.AccelerationDesired := Block.parameters.Motor.rAcceleration;
	MotorDriveUnit.Calculation := CALC_ACC_PULSES;
	MotorDriveUnit();
	AxisBK.Parameter.Acceleration := MotorDriveUnit.pulsesAccelerationDesired;

	//AxisBK.Parameter.Deceleration:=	250000;
	MotorDriveUnit.DecelerationDesired := Block.parameters.Motor.rDeceleration;
	MotorDriveUnit.Calculation := CALC_DEC_PULSES;
	MotorDriveUnit();
	AxisBK.Parameter.Deceleration := MotorDriveUnit.pulsesDecelerationDesired;

	//Change manual Speed
	IF xChangeMotorSpeedUp OR xChangeMotorSpeedDown THEN
		MotorDriveUnit.JogSpeedDesired := 2.0;
	ELSE
		MotorDriveUnit.JogSpeedDesired := Block.parameters.Motor.rDriveManSpeed;
	END_IF

	MotorDriveUnit.Calculation := CALC_JOGSPEED_PULSES;
	MotorDriveUnit();
	AxisBK.Parameter.JogSpeed := MotorDriveUnit.pulsesJogSpeedDesired;

	// Speed paramter for auto movements
	MotorDriveUnit.SpeedDesired := Block.parameters.Motor.rDriveAutoSpeed;
	MotorDriveUnit.Calculation := CALC_SPEED_PULSES;
	MotorDriveUnit();
	AxisBK.Parameter.Speed := MotorDriveUnit.pulsesSpeedDesired;

	// Homing: Reference Position
	MotorDriveUnit.HomePositionDesired := Block.parameters.Motor.rReferencePosition;
	MotorDriveUnit.Calculation := CALC_HOMEPOS_PULSES;
	MotorDriveUnit();
	AxisBK.Parameter.HomePosition := MotorDriveUnit.pulsesHomePositionDesired ; // Tranfer in parameter structure

	//Removed the edgepos. It is possible because Block is executed more than x2 lower than axis
	IF xMotorAbsMovOrder AND AxisBK.Status.HomeOK THEN
		AxisBK.Command.Move.Absolute:= TRUE;
		xMotorAbsMovOrder := FALSE;

		// Move absolute counter
		Block.Lg.diMoveAbsCounter:= Block.Lg.diMoveAbsCounter+1;
		LogVertMovementOrder;
	END_IF

	// Block.commands.xBarHomeOrder comes from kernel2Sw and directo to axis
	// Home order
	AxisBK.Command.Home:= EDGEPOS(xMotorHomeOrder);

	AxisBK.Command.Reset:= ((AxisBK.Status.ErrorID<>0) OR AxisBK.Status.PLCopenState.ErrorStop) AND Block.commands.xReset;
	AxisBK.Command.ErrorAcknowledge:= ((AxisBK.Status.ErrorID<>0) AND Block.commands.xReset) OR
										(AxisBK.Status.ErrorID=6023) OR
										(AxisBK.Status.ErrorID=29216) OR
										(AxisBK.Status.ErrorID=5001) OR
										(AxisBK.Status.ErrorID=29207) ;

END_ACTION
```

#### ReadmeBlock.txt - Block package instructions
```
	(* From efi Cretaprint Almazora Castellon

	Block Manager....
	This cyclic task is managing the mapping configuration for all inks system installed on block structure
	Ink systems are controlled by softare commands direcly but are installed with a mapping inside block
	Block Manager mainly consists in sequencial actions as alarms, logic control, Block states, Input Params Motors
	For setting states of block is implemented BlockStatesCtrl
	For contorling movements of block is implemented LogicControl

	ControlStates is pending to remove
	*)
```

#### LocalFunctions.fun
```iecst
FUNCTION AllDevicedStopped : BOOL
	VAR_INPUT
		Block : REFERENCE TO SimpleBlock;
		AxisBK : REFERENCE TO AxisCtrl_typ;
	END_VAR
END_FUNCTION
```

#### BlockCtrl.var - Local variables
```iecst
VAR
	TNotPrinterZero : TON;
	ars_AlrSafetySystemInBlock : AutoResetSound;
	ars_DriveAlarm : AutoResetSound;
	ars_AlrComBarMtr : AutoResetSound;
	ars_BrokenReferSensor : AutoResetSound;
	AxisBK : REFERENCE TO AxisCtrl_typ;
	xMotorHomeOrder : BOOL;
	xCapOrder : BOOL;
	xMotorAbsMovOrder : BOOL; (*Just to Raise the order. It is reseted once sent the information to the Axis*)
	xAnyManualMov : BOOL;
	xOrderToPrint : BOOL;
	xAnyManualMovement : BOOL;
	xStoppedByExcessiveTimeActive : BOOL;
	rCalcPosDesPrint : REAL;
	rMotorAbsPosDesired : REAL; (*Position in mm*)
	rMotorCurrentPos : REAL; (*Position in mm*)
	iLastState : INT;
	nState : INT := 0;
	Block : REFERENCE TO SimpleBlock;
	SimpleBlockAlarmsReseted : SimpleBlock_Alarms;
	SimpleBlockAlarmsSummaryReseted : stEFI_AlarmSummary;
	T_SafetyError : TOF;
	TON_excessiveBlockActivated : TON;
	T_DelayAlarmRef : TON;
	iTimesStopMovWhileHoming : UINT;
	iTimesStateBlockGoingToPrint : USINT;
	iTimesStateBlockUndefined : USINT;
	iTimesStateBlockPrinting : USINT;
	iTimesStateBlockGoingToCap : USINT;
	iTimesStateBlockInCap : USINT;
	iTimesStateBlockHomingBar : USINT;
	MotorDriveUnit : DriveUnitMngr;
	iReasonStop : UDINT;
	iReasonCritical : UDINT;
	VerMotorEventLog : EventLog_typ;
	stEventLog : EventLog_typ;
	strAuxEventDesc : STRING[129];
	xChangeMotorSpeedUp : BOOL; (*Signal to change motor speed in manual up movements by near limit*)
	xChangeMotorSpeedDown : BOOL; (*Signal to change motor speed in manual down movements by near limit*)
	TON_DelayAnyDriveAlarm : TON;
	ars_EmergencyStop : AutoResetSound;
	BlockStatePrevious : Block_States_enum;
	MachineStatePrevious : enumEFI_GenMachineState;
	BlockPositionPrevious : Block_Position_enum;
	iReasonMovingMan : UINT;
	xBlockPosChange : BOOL;
	xInCap : BOOL; (*Internal var to define if the block is in this position*)
	xInPrint : BOOL; (*Internal var to define if the block is in this position*)
	iReasonAnyWarning : UINT;
	iReasonSafetyGeneral : UINT;
	iCancelHomingBar : UINT;
END_VAR
```

### Program Logical/ExtPack/SimpleBlockCtrl/SimpleBlockCtrl_v1/InitSimpleBlockCtrl (IEC)

#### InitiSimpleBlockCtrl.st
```iecst
PROGRAM _CYCLIC
	gIndexSimpleBlock:= 1;
END_PROGRAM
```

### Program Logical/ExtPack/SimpleBlockCtrl/SimpleBlockSim/SimpleBlockSim_v1/SimpleBlockSim (IEC)

#### Main.st - Init, cyclic, exit code
```iecst
PROGRAM _CYCLIC
	(* Insert code here *)

	Block ACCESS ADR(gSimpleBlock[iSimpleBlockSimIndex]);
	MotorBlock  ACCESS ADR (gAxis[Block.parameters.iMotorAxisIndex]);
	SimBlock ACCESS ADR (gSimSimpleBlock[iSimpleBlockSimIndex]);

	//Managing the homing of the Elevation motor
	IF EDGEPOS(MotorBlock.Status.PLCopenState.Homing AND NOT SimBlock.Commands.DelayHomingBar ) THEN
		iRefSignalState:=1;
		TimesExcecHoming:=TimesExcecHoming+1;
	END_IF

	StatusNcAccess := ncaccess(ncACP10MAN, ADR(MotorBlock.Parameter.Init.AxisObjectName), ADR(AxisRef));

	fbWriteRefSignal.Axis := AxisRef;
	fbWriteRefSignal.ParID := ACP10PAR_VAR_I4_0;
	fbWriteRefSignal.DataType := ncPAR_TYP_DINT;
	fbWriteRefSignal.DataAddress := ADR(uiValueRef);

	CASE iRefSignalState OF
		0:
			fbWriteRefSignal.Execute := FALSE;
		1:
			//IF EDGEPOS(iRefSignalState=2) THEN fbWriteRefSignal.Execute := TRUE; END_IF
			IF NOT fbWriteRefSignal.Done AND NOT fbWriteRefSignal.Busy THEN
				fbWriteRefSignal.Execute := TRUE;
			END_IF
			uiValueRef:=1;
			IF fbWriteRefSignal.Done THEN
				fbWriteRefSignal.Execute := FALSE;
				iRefSignalState:=2;
			END_IF

		2:
			//IF EDGEPOS(iRefSignalState=2) THEN fbWriteRefSignal.Execute := TRUE; END_IF
			IF NOT fbWriteRefSignal.Done AND NOT fbWriteRefSignal.Busy THEN
				fbWriteRefSignal.Execute := TRUE;
			END_IF
			uiValueRef:=0;
			IF fbWriteRefSignal.Done THEN
				fbWriteRefSignal.Execute := FALSE;
				iRefSignalState:=3;
			END_IF

		3:
			//IF EDGEPOS(iRefSignalState=2) THEN fbWriteRefSignal.Execute := TRUE; END_IF
			IF NOT fbWriteRefSignal.Done AND NOT fbWriteRefSignal.Busy THEN
				fbWriteRefSignal.Execute := TRUE;
			END_IF
			uiValueRef:=1;
			IF fbWriteRefSignal.Done THEN
				fbWriteRefSignal.Execute := FALSE;
				iRefSignalState:=0;
			END_IF

	END_CASE

	fbWriteRefSignal();

	iSimpleBlockSimIndex:= iSimpleBlockSimIndex + 1;

END_PROGRAM
```

### Package Logical/GStructs - Global Types

### General.typ - Global General data types
```iecst
TYPE
	TimeStatus_enum :
		(
		TIME_NOT_INITIALIZED,
		TIME_SETTING_TIMEZONE,
		TIME_SETTING_CLIENT,
		TIME_GETTING_TIMEDATA,
		TIME_RECEIVING_DATA,
		TIME_IDLE
		);
	CardType_enum :
		(
		CARD_UNDEFINED,
		CARD_X1, (*First embebed card in CPU 1382*)
		CARD_X2, (*Second embebed card in CPU 1382*)
		CARD_X3, (*Third embebed card in CPU 1382*)
		CARD_CPU1382,
		CARD_CPU0483,
		CARD_CPU0484,
		CARD_DI16,
		CARD_DO16,
		CARD_AI2,
		CARD_AI4,
		CARD_AI8,
		CARD_AO2,
		CARD_AO4,
		CARD_AO8,
		CARD_AT2,
		CARD_AT4,
		CARD_PS33, (*Power Supply Card*)
		CARD_SM, (*Stepper Motor Card*)
		CARD_SC, (*Safety Card SC*)
		CARD_SL, (*Safety Card SL*)
		CARD_SI, (*Safety Input Card*)
		CARD_SO, (*Safety Output Card*)
		CARD_BC (*Coms Card*)
		);
	CardRequiredType_enum :
		(
		CARDREQUIRED_UNDEFINED, (*Defaul value. Used to determine the end of the list*)
		CARDREQUIRED_ALWAYS,
		CARDREQUIRED_ANALOG_THICK,
		CARDREQUIRED_SENSOR_THICK,
		CARDREQUIRED_VACUUM,
		CARDREQUIRED_LED_WHITE,
		CARDREQUIRED_LED_COLOR,
		CARDREQUIRED_HEATED_TANKS,
		CARDREQUIRED_PBF
		);
	PlcCardMapping : 	STRUCT
		Status01 : USINT;
		Status02 : USINT;
		ModuleOk : BOOL;
		DInput : ARRAY[1..MAX_LAST_SIGNAL]OF BOOL;
		DOutput : ARRAY[1..MAX_LAST_SIGNAL]OF BOOL;
		AInput : ARRAY[1..MAX_LAST_SIGNAL]OF INT;
		TempInput : ARRAY[1..MAX_LAST_SIGNAL]OF INT;
		AOutput : ARRAY[1..MAX_LAST_SIGNAL]OF INT;
		CountInput : ARRAY[1..MAX_LAST_SIGNAL]OF UINT;
		ShowTexts : BOOL;
	END_STRUCT;
	StSiUnit : 	STRUCT
		ModuleOk : BOOL;
		NodeStatus : UINT;
		Input01_08 : USINT;
		Input09_16 : USINT;
		Input17_24 : USINT;
		Input25_32 : USINT;
		Output01_08 : USINT;
		Output09_16 : USINT;
		Output17_24 : USINT;
		Output25_32 : USINT;
	END_STRUCT;
	StSiUnitPwrLnk : 	STRUCT
		ModuleOk : BOOL;
		NodeStatus : UINT;
		Input01_16 : UINT;
		Input17_32 : UINT;
		Input33_48 : UINT;
		Input49_64 : UINT;
		Output01_16 : UINT;
		Output17_32 : UINT;
		Output33_48 : UINT;
		Output49_64 : UINT;
	END_STRUCT;
	MachineAutoLocation_enum :
		(
		MACHLOC_UNDEFINED,
		MACHLOC_LOCAL,
		MACHLOC_REMOTE
		);
	UPS_Inputs : 	STRUCT
		xPowerFault : BOOL;
		xByPass : BOOL;
		xLowBattery : BOOL;
		xSystemFault : BOOL;
		xInverterFailure : BOOL;
		xGeneralAlarm : BOOL;
		xUtilityFailure : BOOL;
		LoadOnUtility : BOOL;
		LoadOnBattery : BOOL;
	END_STRUCT;
	plcVersion : 	STRUCT
		iVersion0 : UINT;
		iVersion1 : UINT;
		iVersion2 : UINT;
		iVersion3 : UINT;
	END_STRUCT;
	TestExecution : 	STRUCT
		xSimMachine : BOOL; (*Active if the current machine is simulated and tests are enabled*)
		xAnyTestActive : BOOL;
		TestName : STRING[80];
		iTestState : USINT;
		TestStateDesctiption : STRING[80];
		testPassedAsserts : UDINT;
		testFailedAsserts : UDINT;
		xSometestFailedAsserts : BOOL;
	END_STRUCT;
	TimeMachineParameters : 	STRUCT
		UTCTimeZone : INT; (*Define the UTC time zone of the allocation*)
		DayLightSavingsTime : BOOL; (*Define if the DayLight saving time is active in the allocation*)
	END_STRUCT;
	TimeMachineStatus : 	STRUCT
		LastError : UINT;
		SwState : UINT;
		TimeUpdated : BOOL; (*Time updated by the NtpServer*)
	END_STRUCT;
	TimeMachine : 	STRUCT
		Params : TimeMachineParameters;
		State : TimeStatus_enum;
		Status : TimeMachineStatus;
	END_STRUCT;
	PLCCardDataTexts : 	STRUCT
		Details : STRING[80]; (*Content related*)
	END_STRUCT;
	PLCCardDataStatus : 	STRUCT
		ViewTexts : ARRAY[0..16]OF BOOL; (*Active if there are text assigned*)
		Content : STRING[80]; (*Content related*)
	END_STRUCT;
	PLCCardData : 	STRUCT
		pCard : UDINT; (*Pointer to the card*)
		stCardName : STRING[80]; (*Caed name to show in diagnostic*)
		Type : CardType_enum := CARD_UNDEFINED; (*PLC Card Type*)
		RequiredForFunctions : ARRAY[0..MAX_LAST_REQUIRED_FUNCTION_CARD]OF CardRequiredType_enum := [4(CARDREQUIRED_UNDEFINED)];
		Texts : ARRAY[0..16]OF PLCCardDataTexts; (*Element 0 is not used*)
		Status : PLCCardDataStatus;
		Location : PLCCardLocation;
	END_STRUCT;
	PLCCardLocation :
		(
		CardInPDC,
		CardInPrinter
		);
END_TYPE
```

### GeneralMachine.typ - Global General Machine data types
```iecst
TYPE
	CommsType_enum :
		(
		NoCommsType,
		Type_OpcUa,
		Type_ModbusTcp
		);
	MachineModel_enum :
		(
		NoType,
		Type_P4_12B,
		Type_P4_6B,
		Type_P4_12B_L,
		Type_P4_6B_L,
		Type_SHLD,
		Type_SHLD_L,
		Type_S1400,
		Type_S1400_VAC_PWRLNK,
		Type_S1400_VAC_CAN,
		Type_NOZ_2_AQ,
		Type_P5_OIL,
		Type_P5_WTR,
		Type_P4_CBK,
		Type_NOZ_2_UV,
		Type_NOZ_2_UV_White,
		Type_CUBE_INSPECTION,
		Type_CUBE,
		Type_CUBE_GULLIVER_INSPECTION,
		Type_CUBE_GULLIVER,
		Type_MECANO_UV_WHITE,
		Type_MECANO_UV_OPV,
		Type_MECANO_UV_WHITE_OPV
		);
	CleaningBeltState_enum :
		(
		CLN_BELT_NOT_READY := 0, (*System not ready to execute a clean belt process*)
		CLN_BELT_READY_TO_CLEAN := 1, (*System ready to execute a clean belt process*)
		CLN_BELT_CLEANING_START := 2, (*Starting printer's belt movement at clean belt speed defined by Sw*)
		CLN_BELT_CLEAN_CLOKWISE := 3, (*Start brushes to move clockwise*)
		CLN_BELT_CLEAN_COUNTERCLOCKWISE := 4, (*Start brushes to move counterclockwise*)
		CLN_BELT_CLEANED := 5,
		CLN_BELT_ERROR := 6
		);
	CleaningState_enum :
		(
		CLN_NOT_CLEANING := 1,
		CLN_LINEDELAYING_GAP := 2,
		CLN_READY_TO_CLEAN := 3,
		CLN_CLEANING_ALL_START := 4,
		CLN_CLEANING_ALL_CLEANING := 5,
		CLN_CLEANING_1_START := 6,
		CLN_CLEANING_1_CLEANING := 7,
		CLN_CLEANING_BTW_BLOCKS := 8,
		CLN_CLEANING_2_START := 9,
		CLN_CLEANING_2_CLEANING := 10,
		CLN_CLEANING_JUST1_START := 11,
		CLN_CLEANING_JUST1_CLEANING := 12,
		CLN_CLEANING_JUST2_START := 13,
		CLN_CLEANING_JUST2_CLEANING := 14
		);
	MachineLights_enum :
		(
		MACHINE_LIGHTS_NOT_DEFINED,
		MACHINE_LIGHTS_BEACON,
		MACHINE_LIGHTS_RGB
		);
	ProductDetectSignal_enum :
		(
		PDCFG_NOT_DEFINED,
		PDCFG_SENSOR,
		PDCFG_CARRIAGE,
		PDCFG_SENSOR_AND_CARRIAGE
		);
	StartUpStatus_enum :
		(
		STRUP_DISABLED,
		STRUP_NOT_STARTED,
		STRUP_RESETTING_MOTORS,
		STRUP_HOME_ICLA_ORDER,
		STRUP_HOMING_ICLA,
		STRUP_MOVING_TRAY_OUT,
		STRUP_HOMING_BLOCK,
		STRUP_BLOCK_GOING_TO_CAP,
		STRUP_STARTING_INKS,
		STRUP_WAIT_INKS_STARTED,
		STRUP_REVIEWING_INKS,
		STRUP_POWER_UP_PRINTHEADS,
		STRUP_REVIEWING_PRINTHEADS,
		STRUP_ERROR,
		STRUP_READY,
		STRUP_CANCELLED
		);
	StGeneral_CleanBeltInputs : 	STRUCT
		xLowPosition : BOOL; (*This sensor is active when cylinder is fully in low position.*)
		xHighPosition : BOOL; (*This sensor is active when brush is in place*)
		xError : BOOL; (*The motor relay controls the voltage and current of the motor. If relay is in fault state, this signal will be active*)
		xOpenGuide : BOOL; (*TRUE when clean belt system is not in position*)
	END_STRUCT;
	StGeneral_ProductDetectInputs : 	STRUCT
		pPDCarriageSignalL1 : UDINT; (*Pointer to ProductDetect Signal coming from the Carriage Board*)
		pPDCarriageSignalL2 : UDINT; (*Pointer to ProductDetect Signal coming from the Carriage Board*)
		pPDCarriage2SignalL1 : UDINT; (*Pointer to ProductDetect Signal coming from the Carriage Board 2*)
		pPDCarriage2SignalL2 : UDINT; (*Pointer to ProductDetect Signal coming from the Carriage Board 2*)
		pPDSignalSensorL1 : UDINT; (*Pointer to ProductDetect Signal coming directly from the sensor*)
		pPDSignalSensorL2 : UDINT; (*Pointer to ProductDetect Signal coming directly from the sensor*)
		xAnalogSignalError : BOOL;
		iAnalogSignal : INT;
	END_STRUCT;
	stGeneral_Inputs_Sw : 	STRUCT  (*All this commands are Edge commands*)
		xStart_GI : BOOL; (*EDGE*)
		xStop_GI : BOOL; (*Edge command*)
		xMute_GI : BOOL; (*EDGE*)
		xPause_GI : BOOL; (*EDGE*)
		xReset_GI : BOOL; (*EDGE*)
		xToStop_GI : BOOL; (*Edge commandBool to Stop Mode*)
		xToNormal_GI : {REDUND_UNREPLICABLE} BOOL; (*Edge commandBool to start AutoRun Mode*)
		xToLaboratory_GI : BOOL; (*Edge commandBool to Laboratory Mode*)
		xToByPass_GI : BOOL; (*Edge commandBool to start Bypass Mode*)
		xToJamRecovery : BOOL; (*Edge commandBool to start JamRecovery Mode*)
		xRushProof : BOOL; (*SW marks media to be rejected*)
		xCleanBelt : BOOL; (*SW will active this command when asking a belt cleaning*)
		xCancelStartUp : BOOL; (*SW will active this command when asking to cancel StartUp*)
	END_STRUCT;
	StGeneral_Inputs_Buttons : 	STRUCT  (*Buttons and selectors*)
		xStart : BOOL; (*EDGE*)
		xStop : BOOL; (*EDGE*)
		xManual : BOOL;
		xZero : BOOL;
		xAuto : BOOL;
		xReset : BOOL;
		xMute : BOOL;
	END_STRUCT;
	StGeneral_Inputs : 	STRUCT
		Buttons : StGeneral_Inputs_Buttons;
		x24Vdc : BOOL;
		x230V : BOOL;
		UPSs : ARRAY[0..2]OF UPS_Inputs; (*Element 0 is not used*)
		xConsentL1Ok : BOOL;
		xConsentL2Ok : BOOL;
		xExternalCleaningOrder : BOOL;
		xPC1Ok : BOOL;
		xPC2Ok : BOOL;
		xAirSupply : BOOL; (*General air supply pressure  (ok = TRUE)*)
		iMachineModelCode : INT;
		xSafetyEnabled : BOOL; (*From Safety program*)
		xPbfCardOK : BOOL;
		iRelieve1 : UINT;
		iRelieve2 : UINT;
		xTankHeaterPsuOK : BOOL; (*Signal when Just 1 PSU for TankHeating in the machine*)
		xCoolingPCSensorAlrm : BOOL;
		xCameraDefectDetected : BOOL;
		xRemoteReset : BOOL; (*Reset order in machine remotely controlled*)
		xRemoteJog : BOOL; (*Jog order in machine remotely controlled*)
		CleanBelt : StGeneral_CleanBeltInputs;
		ProductDetect : StGeneral_ProductDetectInputs;
		xDegasserPressure : BOOL;
		xHoppersSoftStarterFault : BOOL;
		xOvervoltage : BOOL;
		xPowerSwitch : BOOL := TRUE; (*Power switch located on printer's cabinet door*)
		xWasteInkTankMaxLevelReached : BOOL;
		AntiStatic : StGeneral_AntiStatictInputs;
	END_STRUCT;
	StGeneral_AntiStatictInputs : 	STRUCT
		xIonLevelAlarm : BOOL; (*Wastage of the antistatic device electrodes*)
		xGenAlarm : BOOL; (*General malfunction alarm of the antistatic device*)
	END_STRUCT;
	StGeneral_Camera_Params : 	STRUCT
		xInstalled : BOOL;
		iMappingBar : USINT;
	END_STRUCT;
	StGeneral_Camera_OrdersSw : 	STRUCT
		xCalibration : BOOL; (*Camera's calibrations process activated*)
	END_STRUCT;
	StGeneral_Camera : 	STRUCT
		Parameters : StGeneral_Camera_Params;
		OrdersSw : StGeneral_Camera_OrdersSw;
	END_STRUCT;
	StGeneral_AirCleaner : 	STRUCT
		Parameters : StGeneral_AirCleaner_Parameters;
		OrdersSw : StGeneral_AirCleaner_SwOrders;
		ParSw : StGeneral_AirCleaner_ParSw;
		Alarms : StGeneral_AirCleaner_Alarms;
	END_STRUCT;
	StGeneral_AirCleaner_Alarms : 	STRUCT
		xDriveComms : BOOL;
		xInverterPowerFault : BOOL;
		xBlowerNotRunning : BOOL;
		xDriveError : BOOL;
	END_STRUCT;
	StGeneral_AirCleaner_SwOrders : 	STRUCT
		xRun : BOOL; (*Delay time before turning off the turbine in auto mode*)
	END_STRUCT;
	StGeneral_AirCleaner_ParSw : 	STRUCT
		rDutyCycle : REAL; (*Speed in %*)
	END_STRUCT;
	StGeneral_AirCleaner_Parameters : 	STRUCT
		iIndex : USINT;
		Direction : MotorDirection_enum;
		xInstalled : BOOL;
		rMaxSpeed : REAL;
	END_STRUCT;
	StGeneral_ApplicationBar : 	STRUCT
		xInstalled : BOOL;
		xDebugMode : BOOL;
		xEnableToPrint : BOOL;
	END_STRUCT;
	StGeneral_HwData : 	STRUCT
		xSimulation : BOOL; (*Defines if the machine is a Simulator*)
		Family : USINT;
		Name : STRING[20];
		SerialNumber : STRING[80]; (*Serial number of the machine*)
		xIsWater : BOOL;
		xIsCubik : BOOL;
		xIsPlatform5 : BOOL; (*Is machine platform 5 to software*)
		xUpsOutOfPrinter : BOOL; (*This printer has no UPS in its cabinet*)
	END_STRUCT;
	StGeneral_Excutions : 	STRUCT
		slow : UDINT;
		fast : UDINT;
	END_STRUCT;
	StGeneral_States_Inks : 	STRUCT
		xAnyStarted : BOOL; (*Any Ink System started*)
		rMaxTempSetPoint : REAL; (*Maximum SetPoint for Started systems*)
		rMinTempSetPoint : REAL; (*Minimum SetPoint for Started systems*)
		rMaxTemp : REAL; (*Maximum Temperature for Started Systems*)
		rMinTemp : REAL; (*Minimum Temperature for Started Systems*)
	END_STRUCT;
	StGeneral_States_Consent : 	STRUCT
		xConsent : BOOL; (*Internal bool used on printer to set state in CONSENT printer*)
		xLackOfConsent : BOOL; (*Machine has order to move the Belt but it is stooped because there is no consent in the line*)
		xUpWithNoConsent : BOOL;
		xUpWithNoConsentCountingTime : BOOL; (*The timer for xUpWithNoConsent is counting*)
		xOrderToEmpyBelt : BOOL; (*The  Belt has to be emptyed, so started the belt without consent*)
	END_STRUCT;
	StGeneral_States_Position : 	STRUCT
		xGoingToPrint : BOOL; (*Internal bool used on printer to set state NOT CAP/NOT PRINT in printer*)
		xInPrint : BOOL; (*Internal bool used on printer to set state PRINTING in printer*)
		xCleaning : BOOL; (*Internal bool used on printer to set state CLEANING in printer*)
		xGoingToCap : BOOL; (*Internal bool used on printer to set state NOT CAP/NOT PRINT in printer*)
		xInCap : BOOL; (*Internal bool used on printer to set state CAPPED in printer*)
	END_STRUCT;
	StGeneral_States_ProductDetect : 	STRUCT
		xProductDetectL1 : BOOL; (*Any product detect in L1. In any line and coming from Carriage or Sensor directly. It means that a media has been printed*)
		xProductDetectL2 : BOOL; (*Any product detect in L2. In any line and coming from Carriage or Sensor directly. It means that a media has been printed*)
		xAnyProductDetect : BOOL; (*Any product detect. In any line and coming from Carriage or Sensor directly. It means that a media has been printed*)
		xAnyProductDetectDtpStricted : BOOL; (*Any product detect. In any line and coming from Carriage or Sensor directly. Refused L2 if not in DTP*)
	END_STRUCT;
	StGeneral_States_Remote : 	STRUCT
		xMachineReady : BOOL; (*Machine in Print position with Blowers and Belt ready*)
		xReadyToJogInJamRecovery : BOOL; (*Bars in safety print position and ready to receive the jog order*)
		xSafetyReadyToReset : BOOL; (*Safety ready to be reseted*)
		xBeltNotStopped : BOOL; (*The signal is always TRUE, and when the belt stops, it is reseted during a second*)
	END_STRUCT;
	StGeneral_States_CleaningBelt : 	STRUCT
		enState : CleaningBeltState_enum;
		xCleaningProcessOnGoing : BOOL; (*Clean belt process is being executed*)
		TimeDelaySwapDirBeltCleanMotor : TIME; (*Time to wait before swap belt clean motor direction*)
		xCleanRequired : BOOL; (*Clean belt process must be executed*)
		iTimeToCleanBelt : INT;
	END_STRUCT;
	StGeneral_States_Cleaning : 	STRUCT
		enCleaningState : CleaningState_enum;
		iCleaningState : UINT; (*Cleaning State value to Sw*)
		xCleanRequestToLine : BOOL; (*When an internal cleaning request is set and machine is controlled by line*)
		xCleanRequired : BOOL; (*The printer will clean automatically in less than 10' when this signal is activated*)
		xCleanInminent : BOOL; (*The printer will clean automatically in 30" after this signal is activated. SendJob should be lowered and not raised*)
		MinutesInStopForClean : UDINT; (*Software Output*)
		MinutesInProdForClean : UDINT; (*Software Output*)
		MinutesForClean : UDINT; (*Software Output*)
		MinutesTotalTimeForClean : UDINT; (*Software Output*)
		iPieceCounterBtwCleaningsL1 : INT;
		iPieceCounterBtwCleaningsL2 : INT;
	END_STRUCT;
	StGeneral_States_Blocks : 	STRUCT
		xBlockAlarmToEmpyBelt : BOOL; (*An alarm in a block is detected asking to Empty Belt*)
		xAnyPrintheadPowered : BOOL; (*Internal state to heater tanks used on alarm PSU*)
		xAnyTankHeaterEnabled : BOOL; (*Internal state to heater tanks used on alarm PSU*)
		xAnyBlockToPrint : BOOL;
		xAnyBarAndBlockReadyToPrint : BOOL;
	END_STRUCT;
	StGeneral_States_StartUp : 	STRUCT
		Status : StartUpStatus_enum;
		xReadyToAuto : BOOL; (*The startup process has finish and the machine is ready to Auto*)
		xInProgress : BOOL;
	END_STRUCT;
	StGeneral_States_MountedMedia : 	STRUCT
		rOverThicknessToMounted : REAL; (*The value to consider Mounted media depending on the speed*)
	END_STRUCT;
	StGeneral_States : 	STRUCT
		Position : StGeneral_States_Position;
		Mode : StGeneral_States_Mode;
		Consent : StGeneral_States_Consent;
		ProductDetect : StGeneral_States_ProductDetect;
		Remote : StGeneral_States_Remote;
		Cleaning : StGeneral_States_Cleaning;
		CleaningBelt : StGeneral_States_CleaningBelt;
		Inks : StGeneral_States_Inks;
		Blocks : StGeneral_States_Blocks;
		Clear : StGeneral_ApplicationBar;
		Color : StGeneral_ApplicationBar;
		White : StGeneral_ApplicationBar;
		StartUp : StGeneral_States_StartUp;
		MountedMedia : StGeneral_States_MountedMedia;
		xBeltRunPrevToClean : BOOL; (*Internal state in printer used on gap and delay line*)
		iAutoModeSW : INT; (*Printer State to sw *)
		iMachineModelCodeSW : INT; (*Printer model to Sw, in function of HW ID code*)
		StateMode : enumEFI_GenMachineState; (*states*)
		AutoMode : stEFI_MachineAutoModes; (*commands*)
		uiLicenseCounter : UINT;
		xStarted : BOOL; (*TRUE if the PLC is running*)
		exec : StGeneral_Excutions;
		HwData : StGeneral_HwData;
		iFaultRunPlc : INT; (*Software Output ??*)
		xMediaDetected : BOOL; (*Media detected before product detect. Detected in Analog or in 3sensors*)
		xRobotReadyToPrint : BOOL;
		xWorkingAsPBF : BOOL; (*An indication of working as PBF is received*)
		iJamDevices : USINT := 0; (*Quantity of Jam Devices installed in the machine*)
		xAbortJobRequest : BOOL;
		xProtectBendedWithPause : BOOL; (*Increase the height of the media inside the machine to protect the printheads*)
		xDoubleLineAllowed : BOOL; (*Machine allows double line printing (depending on objects enabled and line configuration)*)
	END_STRUCT;
	StMachine_ConstantParameters : 	STRUCT
		rMinTicknessMedia : REAL; (*mm*)
		rMaxTicknessMedia : REAL; (*mm*)
		rMountedMediaLevelInBypassMode : REAL; (*mm*)
		rMaxMountedPieceOverThick : REAL; (*Max value in mm to consider a piece as mounted piece*)
		rMinMountedPieceOverThick : REAL; (*Minimum value in mm to consider a piece as mounted piece*)
		rMinMarginPrinting : REAL; (*mm*)
		rMaxMarginPrinting : REAL; (*mm*)
		rDistanceBeltInitToPd : REAL; (*Distance Between belt init to PD Sensor (mm)*)
		rDistanceThicknesToPD : REAL; (*Distance Between Thicknes Detection To PD Sensor (mm)*)
		iNumBlocks : USINT; (*For writting the number of blocks in a machine*)
		iNumTransVacuum : USINT; (*For writting the number of TransportVacuum in a machine*)
		iNumCuringLeds : USINT; (*Total curing modules in machine*)
		iNumSensorsPerJamDevice : USINT := 4; (*For writing the number of Sensors in each Jam Device*)
		iNumSAIInstalled : USINT; (*Number of SAI installed in machine*)
	END_STRUCT;
	StGeneral_CleanBeltTopPar : 	STRUCT
		xCleanBeltContinue : BOOL; (*Input software parameter from Sw*)
		xCleanBeltByTiles : BOOL; (*Input software parameter from Sw*)
		xCleanBeltByTime : BOOL; (*Input sw param using time param iCleaningBeltByTime*)
		tiCleaningBeltDuration : TIME; (*Time in seconds. Input software parameter from Sw*)
		tiCleaningBeltByTime : TIME; (*Time in Minutes. Input software parameter from Sw*)
		xCleanBeltForced : BOOL; (*Edge Command. Input software parameter from Sw*)
		iSPTilesToCleanBelt : UINT; (*Input software parameter from Sw*)
	END_STRUCT;
	StGeneral_CleanBeltParameters : 	STRUCT
		xCleanBeltContinue : BOOL; (*Input software parameter from Sw*)
		xCleanBeltByTiles : BOOL; (*Input software parameter from Sw*)
		xCleanBeltByTime : BOOL; (*Input sw param using time param iCleaningBeltByTime*)
		tiCleaningBeltDuration : TIME; (*Time in seconds. Input software parameter from Sw*)
		tiCleaningBeltByTime : TIME; (*Time in Minutes. Input software parameter from Sw*)
		xCleanBeltForced : BOOL; (*Edge Command. Input software parameter from Sw*)
		iSPTilesToCleanBelt : UINT; (*Input software parameter from Sw*)
		xMoveBackward : BOOL;
		xMoveForward : BOOL;
		iBeltTurns : UINT; (*Number of belt turns cleaning the belt. Just used in UV scenario*)
		xTurbineEnabled : BOOL;
		iBeltSpeed : UINT; (*Speed used to clean the belt. Just used in UV scenario*)
	END_STRUCT;
	StGeneral_CleanParameters : 	STRUCT
		iCleaningType : INT; (*0: Undefined, 1:Venturi, 2:Turbine    Is not implemented in Control, pending to get from Schneider this functionality*)
		xCleaningBlocksInSeq : BOOL; (*SoftwareInput New Var*)
		xCleanSystemByTime : BOOL; (*Software Input*)
		xEnableCleaningInStopMode : BOOL;
		iPiecesNumberToCleanL1 : INT; (*SoftwareInput*)
		iPiecesNumberToCleanL2 : INT; (*SoftwareInput*)
		xCleanSystemByPieces : BOOL; (*SoftwareInput *)
		tiTimeDelayToCleanL1 : TIME; (*SoftwareInput*)
		tiTimeDelayToCleanL2 : TIME; (*SoftwareInput*)
		tiTimeDelayGapToClean : TIME; (*SoftwareInput*)
		tiCleaningByTime : TIME; (*SoftwareInput*)
		tiToCleanWhenPrinterStopped : TIME; (*Time in minutes*)
		tiBetweenCleaningBlocks : TIME;
		iCleanMotorSpeedBwd : INT; (*Software Input. *)
		iCleanMotorSpeedFwd : INT; (*Software Input. *)
	END_STRUCT;
	StGeneral_ShotParameters : 	STRUCT
		xShotLine1 : BOOL; (*Edge command bool*)
		xShotLine2 : BOOL; (*Edge command bool*)
		xRepetitionShotLine1 : BOOL; (*State command bool*)
		xRepetitionShotLine2 : BOOL; (*State command bool*)
		tiShotL1 : TIME; (*Input software parameter from Sw*)
		tiShotL2 : TIME; (*Input software parameter from Sw*)
	END_STRUCT;
	StGeneral_CleanBelt : 	STRUCT
		xCleanBeltMoveFwd : BOOL; (*While this signal is active the motor turns clockwise*)
		xCleanBeltMoveBwd : BOOL; (*While this signal is active the motor turns counter-clockwise*)
		xCleanBeltResetRelay : BOOL; (*Reset belt clean motor relay*)
		xCleanBeltPump : BOOL; (* Set pneumatic pump*)
		xCleanBeltTopScraper : BOOL;
		xStart : BOOL; (*To start clean belt*)
		xPistonFlojet : BOOL; (* Set pneumatic piston*)
	END_STRUCT;
	StGeneral_DtpParameters : 	STRUCT
		xDoubleLine : BOOL; (*SoftwareInput*)
		iModeLine1 : INT; (*SoftwareInput. 0=RUN 1=BYPASS 2=STOP*)
		iModeLine2 : INT; (*SoftwareInput. 0=RUN 1=BYPASS 2=STOP*)
	END_STRUCT;
	StGeneral_SuctionParameters : 	STRUCT
		iBlowerMode : INT; (*Suction mode functionality. It can be configured by GUI with Ventrui when is 1 or Turbine when is 2. Parameters received from GUI*)
		tiBlowerDelayOff : TIME; (*Delay time before turning off the turbine in auto mode*)
	END_STRUCT;
	StGeneral_PCsParameters : 	STRUCT
		xExistPC1 : BOOL; (*Software Input Cmd*)
		xExistPC2 : BOOL; (*Software Input Cmd*)
		xKeepPcsOn : BOOL;
	END_STRUCT;
	StGeneral_UI_Parameters : 	STRUCT
		xCriticalCondition : BOOL; (*Sw has a critical alarm not controlled by plc*)
		xWarningCondition : BOOL; (*Sw has a warning alarm not acknowledged by plc*)
		xStartPrintButtonActive : BOOL; (*UI main button displays start print option*)
	END_STRUCT;
	StGeneral_ElectronicsParameters : 	STRUCT
		xPrintServerOK : BOOL; (*Software Input State*)
		xRobotReadyL1 : BOOL; (*SoftwareInput *)
		xRobotReadyL2 : BOOL; (*SoftwareInput*)
		xIsPBF : BOOL;
	END_STRUCT;
	StGeneral_SafetyParameters : 	STRUCT
		rMountedPieceOverthickness : REAL; (*Software Input. Value in mm*)
		rMarginSafePrint : REAL; (*SoftwareInput. Fix offset to bent tile. The heads go to the thickness measured + this value. Value in mm*)
		rMaxBeltSpeedSetPoint : REAL := 70.0; (*Max speed received from gui in m/min*)
	END_STRUCT;
	StGeneral_CuringParameters : 	STRUCT
		xCureBySpeed : BOOL; (*Intensity of lamps set depending on machine speed*)
		xOptimizeCuring : BOOL; (*Curing optmitzation mode required*)
		xCureByStretch : BOOL; (*Curing by stretch mode required*)
	END_STRUCT;
	StGeneral_DocumentParameters : 	STRUCT
		rWidth : REAL; (*Job's document width in mm*)
		rLength : REAL; (*Job's document  length in mm*)
		rOffsetL1 : REAL; (*Job's document offset L1 in mm*)
		rOffsetL2 : REAL; (*Job's document offset L2 in mm*)
	END_STRUCT;
	StGeneral_MediaParameters : 	STRUCT
		rThickness : REAL; (*Tile thickness to print from gui in mm*)
		rWidth : REAL; (*Board's width in mm*)
		rGap : REAL; (*Gap between boards in mm*)
		rLength : REAL; (*Board's length in mm*)
		rOffsetRegisterL1 : REAL; (*Board's offset L1 in mm*)
		rOffsetRegisterL2 : REAL; (*Board's offset L2 in mm*)
	END_STRUCT;
	StGeneral_LampParameters : 	STRUCT
		stSerialNumber : STRING[6];
	END_STRUCT;
	StGeneral_CuringLedParameters : 	STRUCT
		Lamp : ARRAY[0..16]OF StGeneral_LampParameters;
		rPreCuringOffset : REAL := 0.0; (*Pre curing offset set by SW in cm*)
		rPostCuringOffset : REAL := 0.0; (*Post curing offset set by SW in cm*)
	END_STRUCT;
	StGeneral_HwParameters : 	STRUCT
		iMaxNumPowerMeters : USINT := 2; (*Number of chillers allowed by the printer*)
		iMaxNumChillers : USINT; (*Number of chillers allowed by the printer*)
		iMaxCuringLedBars : UINT; (*Number of curing led bars slots allowed by the printer*)
		rMinPrintPosition : REAL; (*Minimum printing position allowed*)
		iWidth : UINT; (*Machine's printing width in mm*)
		xSuctionModeAllowed : BOOL; (*Machine has a mist collector turbine (suction)*)
		xDoubleLineAllowed : BOOL; (*Active when printer allows double line printing*)
	END_STRUCT;
	StGeneral_HwAncillariesParams : 	STRUCT
		xInstallFeeder : BOOL;
		xInstallPrimer : BOOL;
		xInstallDryer : BOOL;
		xInstallOverbarnish : BOOL;
		xInstallStacker : BOOL;
	END_STRUCT;
	StGeneral_HwSetBySwParameters : 	STRUCT
		xInstallThicknessSensor : BOOL; (*Install analog thickness detection system. Active while needed installed*)
		xInstallnSensor : BOOL;
		Ancillaries : StGeneral_HwAncillariesParams;
		iMaxMediaLength : UINT; (*Maximum media length allowed to be loaded in job. In mm*)
	END_STRUCT;
	StGeneral_RemoteParameters : 	STRUCT
		xSendingJob : BOOL; (*A job is been sent by the previous machine. Bars can go to final position*)
	END_STRUCT;
	StGeneral_SwParameters : 	STRUCT
		CleanBelt : StGeneral_CleanBeltParameters;
		CleanBeltTop : StGeneral_CleanBeltTopPar;
		Clean : StGeneral_CleanParameters;
		Shot : StGeneral_ShotParameters;
		Dtp : StGeneral_DtpParameters;
		Suction : StGeneral_SuctionParameters;
		PCs : StGeneral_PCsParameters;
		UI : StGeneral_UI_Parameters;
		Electronics : StGeneral_ElectronicsParameters;
		Safety : StGeneral_SafetyParameters;
		Document : StGeneral_DocumentParameters;
		Media : StGeneral_MediaParameters;
		Hw : StGeneral_HwSetBySwParameters;
		Remote : StGeneral_RemoteParameters;
		Curing : StGeneral_CuringParameters;
		xAutoStartEnabled : BOOL; (*The autostart process is enabled*)
		iFaultComPcPlc : INT; (*Software Input State*)
		rMarginPrint : REAL; (*SoftwareInput, jetting gap in mm*)
		xMachineDirection : BOOL; (*0: Derecha 1: Izquierda*)
		rFirstHeadPosition : REAL;
		rLastHeadPosition : REAL;
		tiDelayConsent : TIME; (*Used on kernel to PLC. Time in seconds*)
		iNumCopies : UDINT; (*Number of boards in a job. Can be changed on the fly.*)
		rBeltSpeedSetPoint : REAL := 20.0; (*Speed in m/min. Input parameter from SW*)
		xDegasser : BOOL;
		xJamDetectEnable : BOOL; (*Jam Detection Enabled*)
	END_STRUCT;
	StGeneral_MediaParams : 	STRUCT
		iMaxMediaWidth : UINT; (*Maximum media width allowed in mm*)
		iMinMediaWidth : UINT; (*Minimum media width allowed in mm*)
		iMaxMediaLength : UINT := 3000; (*Maximum media length allowed in mm*)
		iMinMediaLength : UINT; (*Minimum media length allowed in mm*)
		rMaxMediaThickness : REAL; (*Maximum media thickness allowed in tenths of mm*)
		rMinMediaThickness : REAL; (*Minimum media thickness allowed in tenths of mm*)
	END_STRUCT;
	StGeneral_CleanParams : 	STRUCT
		xEnabledCleanTotalTime : BOOL := FALSE; (*Enabled cleaning machine if total time counted without cleaning. Currently 24h*)
		xCleanBeltTopInstall : BOOL := FALSE; (*Cleanning Belt Scrapper System Installed*)
		xCleanBeltWater : BOOL; (*Cleaning belt system for Noz2 water*)
		xCleanBeltForUv : BOOL := FALSE;
	END_STRUCT;
	StGeneral_VacuumParams : 	STRUCT
		xStartBlowerGoingToPrint : BOOL; (*Start the blowers when in production and going to print*)
		xTransVacuumIndependenParams : BOOL; (*TRUE: Each TransVacuum with different parameters. FALSE: TransVacuum[1] copied to the rest of elements*)
	END_STRUCT;
	StGeneral_CureParams : 	STRUCT
		xCuringByStretchAllowed : BOOL; (*CuringByStretch functionality IS allowed in this machine*)
		xForceMaxWidth : BOOL; (*Force to cure with max width instead of using data from media coming from Sw*)
	END_STRUCT;
	StGeneral_DynMountedMedia : 	STRUCT
		rSpeedMaxMounted : REAL; (*Value in m/min*)
		rSpeedMinMounted : REAL; (*Value in m/min*)
		rMaxOverThickMounted : REAL; (*Value in mm*)
		rMinOverThickMounted : REAL; (*Value in mm*)
	END_STRUCT;
	StGeneral_MountedMedia : 	STRUCT
		Type : ThicknessMountedDetectionType; (*Mounted Type in machine*)
		Dynamic : StGeneral_DynMountedMedia;
		xDynamicMountedMedia : BOOL; (*Configured Dynamic mounted media*)
	END_STRUCT;
	StGeneral_ProductDetectParams : 	STRUCT
		xDisableBrokenSensor : BOOL;
	END_STRUCT;
	StGeneral_Parameters : 	STRUCT
		CT : StMachine_ConstantParameters; (*Printer input constants params*)
		ConfigName : STRING[80];
		ConfigNameID : USINT := 0; (*Identification of the Configuration been executed*)
		CommsType : CommsType_enum; (*Comms protocol used to communicate with kernel*)
		MachineModel : MachineModel_enum; (*HW ID codes are defined here*)
		PDSignalTpe : ProductDetectSignal_enum;
		Media : StGeneral_MediaParams;
		Clean : StGeneral_CleanParams;
		ProductDetect : StGeneral_ProductDetectParams;
		Vacuum : StGeneral_VacuumParams;
		Cure : StGeneral_CureParams;
		MountedMedia : StGeneral_MountedMedia;
		xControlledByLine : BOOL; (*Define if the machine is controlled by a LineManager*)
		xControlledRemotely : BOOL; (*Define if the machine is controlled by an external device. eCommerce*)
		xAllowLaboratory : BOOL; (*Define if the machine allows laboratory behabior or not*)
		xAllowAutoStartUp : BOOL; (*The autostart process is allowed in the machine*)
		xDynamicPrePrintingPos : BOOL; (*The preprinting position is assigned in orders, not in assign data*)
		xJobNotReadyIsCritical : BOOL; (*Active whether machine have to stop when detecting media but no job is ready to be printed*)
		xAllowJamRecovery : BOOL; (*Define if the machine allows JamRecovery behabior or not*)
		xDisableStartHoldingGreenButton : BOOL; (*Disable start production with a long press of Green Button in machine*)
		xLeftHandMachine : BOOL; (*Software Output*)
		xRightHandMachine : BOOL; (*Software Output*)
		rMaxPrintHeadPos : REAL; (*Maxium Print HEad Position to SW in mm*)
		rMinPrintHeadPos : REAL; (*Minium Print HEad Position to SW in mm*)
		xProtectPHForBlowersRunning : BOOL; (*Required to protect the print heads from vacuum drying*)
		tiTimeToRaiseBars : TIME := T#5m; (*Required to protect the print heads from tile bending*)
		xProtectPHWithStoppedMediaBended : BOOL; (*Required to protect the print heads from tile bending*)
		rBeltSpeedWhileEmptyBelt : REAL;
		iMediaFilter : UINT; (*Filter to be used to consider real media detected by PD sensor (Cm)*)
		MachineLights : MachineLights_enum;
		Hw : StGeneral_HwParameters;
	END_STRUCT;
	stGeneral_SerialNumberCommands : 	STRUCT
		xExecute : BOOL; (*EDGE*)
		SerialNumber : STRING[80]; (*Serial number of the machine*)
	END_STRUCT;
	stGeneral_ResetCpuCommands : 	STRUCT
		xExecuteReset : BOOL; (*EDGE*)
		AutorizationCode : STRING[80]; (*Autorization code. h98o76. Deleted after reset*)
	END_STRUCT;
	stGeneral_commandsRemote : 	STRUCT
		xStartBlowers : BOOL; (*Order to Start the blowers. Received from RemoteMachine. It will be falled when out of Auto.Stop*)
	END_STRUCT;
	stGeneral_commands : 	STRUCT
		xAllToCap : BOOL; (*Use as EDGE CommandBool used to send all block to cap. Reseted in program. Line can use it*)
		xAllToPrint : BOOL; (*Use as EDGE CommandBool used to send all block to print. Reseted in program. Line can use it*)
		xResetRouter : BOOL;
		xResetCB : BOOL;
		xResetStrobePdDiff : BOOL; (*Use as EDGE CommandBool. Reseted in program*)
		xCompenserLine1 : BOOL;
		xCompenserLine2 : BOOL;
		xStop : BOOL;
		xRunBelt : BOOL;
		xClean : BOOL;
		ResetCpu : stGeneral_ResetCpuCommands;
		SerialNumber : stGeneral_SerialNumberCommands;
		CleanBelt : StGeneral_CleanBelt;
		Remote : stGeneral_commandsRemote;
	END_STRUCT;
	StGeneral_AutoCommands : 	STRUCT  (*COMMANDS GENERATED INTERNALLY BY CODE, NOT EXTERNALLY*)
		iAutoMode : enumEFI_MachineAutoStatesMode; (*Internal variable to manage AUTOMATIC modes in printer RU,BUPASS, LAB AND STOP*)
		xCleanningByPiecesL1 : BOOL; (*CommandBool state to set cleaning cycle in L1*)
		xCleanningByPiecesL2 : BOOL; (*CommandBool state to set cleaning cycle in L2*)
		xCleanningByExtOrder : BOOL; (*Internal command from external input state to set/enable a cleaning cycle by external order input*)
		xCleanningByTimeProd : BOOL; (*CommandBool state to set cleaning cycle L1 or L2 by time in Production*)
		xCleanningByTotalTime : BOOL; (*CommandBool state to set cleaning cycle by total time after no cleaning*)
		xCleanningByTimeInStopMode : BOOL; (*CommandBool state to set cleaning cycle L1 or L2 by time when block is in cap position*)
		xMuteAlarms : BOOL; (*Edge commandBool used to mute all alarms*)
		xToCap : BOOL; (*Edge commandBool used to send all block to cap*)
		xToPrint : BOOL; (*Edge commandBool used to send all block to print*)
		xReset : BOOL; (*Internal bool used on printer to set state RESET in printer*)
		xStart : BOOL; (*Edge Command to Start the Machine. By button or an specific order from Sw*)
		xStop : BOOL; (*Edge Command to Stop the Machine. By button or an specific order from Sw*)
		xToSafePosition : BOOL; (*ComandBool state to move bars to Safe postion near of print to protect printheads from bended parts or vacuum drying*)
		xCleanModbus : BOOL; (*Order to clean Modbus registers. Usually when a PLC version is detected*)
		xCleanBelt : BOOL; (*Order to clean Modbus registers. Usually when a PLC version is detected*)
	END_STRUCT;
	StGeneral_AlarmsList : 	STRUCT
		xAlrTurbinForCleaning : BOOL; (*Pending to remove in 4.3.6*)
		xAlarmPlarformInc : BOOL; (*AlarmCritical*)
		xAlarmSAIPowerOff : BOOL; (*AlarmCritical - SAI is near to power off*)
		xAlarmAir1 : BOOL; (*AlarmStop*)
		xAlarmComPcPLC : BOOL; (*AlarmStop*)
		xAlarmMountedPiece : BOOL; (*Resume next *)
		xAlarmMountedPieceBypassMode : BOOL; (*AlarmStop*)
		xAlarmNotInPrintPosition : BOOL;
		xAlarmEnableWithoutBarsOn : BOOL;
		xNoActionDangerCollision : BOOL; (*Resume alarms*)
		xNoActionAlarmExist : BOOL; (*Resume alarms*)
		xHeaterTankPsu : BOOL; (*Resume alarms*)
		xPDBrokenSensorL1 : BOOL; (*Product Detect Line 1 Broken or Desconected*)
		xPDBrokenSensorL2 : BOOL; (*Product Detect Line 2 Broken or Desconected*)
		xAlrThicknSystemNotSelected : BOOL; (*Thickness detection system not selected.*)
		xAlarmSAIPowerFault : BOOL; (*Power main suply switch off*)
		xAlr24Vdc : BOOL; (*24VDC Power IDS supply switc off*)
		xAlrWrongPhysConf : BOOL; (*Alarm Critical: Wrong physical configuration or some tarjet are disconected*)
		xAlrDingWrongPosition : BOOL; (*StopAlarm: with product detectt signal without previuos ding signal*)
		xSwCriticalCondition : BOOL; (*Sw is in a critical condition to execute printing process*)
		xNotLoadedImage : BOOL; (*This alarms is an Stop alarm in machines without line. In machines with line, it is a critical alarm for the line*)
		xNoPowered : BOOL; (*This alarm is raised when machine's power switch is not active*)
		xAlrWidthOutLimits : BOOL; (*Parsw media width out of limits*)
		xAlrLengthOutLimits : BOOL; (*Parsw media length out of limits*)
		xAlrThickOutLimits : BOOL; (*Parsw media thickness out of limits*)
		xAlrSafetyNotEnabled : BOOL; (*Printer safety enables nok*)
	END_STRUCT;
	StGeneral_WarningsList : 	STRUCT
		xStopInAuto : BOOL; (*Review*)
		xValidConfiguration : BOOL; (*Review*)
		xSAIFault : BOOL;
		xSAILowBat : BOOL;
		xSAIBypass : BOOL;
		xExternalCleanActive : BOOL;
		xMaxMovsBentTile : BOOL;
		xNotLoadedImage : BOOL; (*Just stopping the belt. Used in ceramics, where we can load image with the belt stopped and restart production*)
		xBentTile : BOOL;
		xPCCabineSensAlrm : BOOL;
		xMountedMediaInside : BOOL;
		xMediaStoppedInside : BOOL;
		xCleanCylinderNotInHighPosition : BOOL;
		xCleanBeltRelayFaulted : BOOL;
		xBeltCleanRequired : BOOL;
		xCleanBeltSystemNotInPosition : BOOL;
		xPbfCardNotOK : BOOL;
		xUpNotConsent : BOOL; (*Resume alarms*)
		xNoCleaningModeEnabled : BOOL; (*Warning: No pressure on degasser circuit*)
		xAlrDegasserPressure : BOOL; (*Warning: No pressure on degasser circuit*)
		xMediaIncoherenceDetectedL1 : BOOL; (*Active when product detect sensor detects media but detection system has not. L1*)
		xMediaIncoherenceDetectedL2 : BOOL; (*Active when product detect sensor detects media but detection system has not. L1*)
		xBeltCleanTurbNotAvail : BOOL; (*VSD ACS380 ok feedback signal not present NOZOMITWO-1912*)
		xWasteInkTankMaxLevelReached : BOOL;
		xOvervoltage : BOOL; (*Warning alarm*)
		xImageLoadedButNoInkBarRelated : BOOL; (*This alarm is raised when image is loaded but no bar has been assigned to that job. Related to status "ColorLoadedInJob"*)
		xErrorAntiStatic : BOOL; (*Antistatic device in error*)
		xIonAntiStatic : BOOL; (*Wastage of the antistatic device electrodes*)
		xAlrHoopersSoftStarterFault : BOOL; (*Warning alarm*)
	END_STRUCT;
	StGeneral_Alarms : 	STRUCT
		Warning : StGeneral_WarningsList;
		Alarm : StGeneral_AlarmsList;
		xAlrDisableGoToProduction : BOOL;
		xAlrSafetySystemEStop : BOOL; (*SLX DI 10 is enable transport from safety progam*)
		xAlarmSound : BOOL;
	END_STRUCT;
	StGeneral_Log : 	STRUCT
		ManualChg : DINT;
		AutoChg : DINT;
		ManualHrs : DINT;
		AutoHrs : DINT;
		VdcHrs : DINT;
		DateStart : DINT;
		udiPiecesCounterErrorL1 : UDINT; (*PD Detection Counter Failed L1*)
		udiPiecesCounterErrorL2 : UDINT; (*PD Detection Counter Failed L2*)
		udiPiecesCounterL1 : UDINT;
		udiPiecesCounterL2 : UDINT;
		diPiecesCounterStrobe : DINT;
		iDiffPiecesStrobeProductDetect : INT; (*Difference of quantity in Product detect signals minus the strobe signals*)
		udiTileCounterBalluffLaser : UDINT; (*Program in mode active..end*)
		udiTileCounterTriggerLaser : UDINT; (*Program in mode active..end*)
		udiDifCounters : UDINT; (*Program in mode active..end*)
		iTilesCounterToClean : UINT;
		iTilesCounterToCleanBeltTop : UINT;
	END_STRUCT;
	StGeneral_Outputs_CleanBelt : 	STRUCT  (*Outputs for cleanbelt*)
		xAirTurbineVSDReset : BOOL; (*Output signal to reset the VSD of the air turbine NOZOMITWO-1912*)
		xAirTurbine : BOOL; (*Output signal to start the air turbine NOZOMITWO-1912*)
	END_STRUCT;
	StGeneral_Outputs : 	STRUCT
		xResetHub : BOOL;
		xResetSwitch : BOOL;
		xResetRouter : BOOL;
		xResetCB1 : BOOL;
		xResetCB2 : BOOL;
		xPC1Start : BOOL;
		xPC2Start : BOOL;
		xRedLight : BOOL;
		xYellowLight : BOOL;
		xWhiteLight : BOOL;
		xBlueLight : BOOL;
		xGreenLight : BOOL;
		xBuzzerButtonPanel : BOOL;
		xConsentL1 : BOOL;
		xConsentL2 : BOOL;
		xCompenserLine1 : BOOL;
		xCompenserLine2 : BOOL;
		xLine1ReadyToClean : BOOL;
		xLine2ReadyToClean : BOOL;
		xSuctionTurbine : BOOL;
		xLightReset : BOOL;
		xAirSupply : BOOL;
		xCoolingPCStart : BOOL;
		iRelief1 : UINT; (*Signal of the Relief readed in line 1*)
		iRelief2 : UINT; (*Signal of the Relief readed in line 2*)
		xShotLine1 : BOOL; (*Output For InstantPrint/ContinuousPrint signal from PLC to Carriage*)
		xShotLine2 : BOOL; (*Output For InstantPrint/ContinuousPrint signal from PLC to Carriage*)
		xRemoteTeachL1 : BOOL;
		xRemoteTeachL2 : BOOL;
		xDegasser : BOOL;
		CleanBelt : StGeneral_Outputs_CleanBelt;
		iTimeBlockAtSafePosition : UINT; (*Counter to acknowledge how many times block has been lifted to safe position*)
		xAntiStaticPOn : BOOL; (*Power on the antistatic device*)
	END_STRUCT;
	StGeneral : 	STRUCT
		In : StGeneral_Inputs;
		St : StGeneral_States;
		Pt : StGeneral_Parameters;
		parSw : StGeneral_SwParameters; (*Software params*)
		commands : stGeneral_commands;
		commandsSw : stGeneral_Inputs_Sw; (*All this commands are Edge commands. Reseted at the end of Machine_Fast*)
		AutoCmd : StGeneral_AutoCommands;
		AlSummary : stEFI_AlarmSummary;
		Al : StGeneral_Alarms;
		Lg : StGeneral_Log;
		Out : StGeneral_Outputs;
	END_STRUCT;
END_TYPE
```

### Package Logical/GVars - Gloval Vars

### Permanents.var
```iecst
VAR RETAIN
	gPermanentSN : STRING[80]; (*Serial Number of the machine*)
	gInksPermanentParBar : ARRAY[0..MAX_LAST_INK] OF stInksBarParams;
	gPermanentInksParSw : ARRAY[0..MAX_LAST_INK] OF stInksParametersSw;
	gPermanentMachine : StGeneral_SwParameters;
	gPermanentBlock : ARRAY[0..MAX_LAST_BLOCK] OF StBlock_SwParameters;
	gPermanentSwBelt : stBelt_SwParameters;
	gPermanentSimMachinePar : SimMachineParameters_typ;
	gPermanentDryer : Dryer_Parameters;
	gPermanentVersion : plcVersion;
	gPermanentTrVacuum : ARRAY[0..MAX_LAST_TRANS_VACUUM] OF TransVacuumParametersSw_typ;
	gPermanentSimpleBlock : SimpleBlock_SwParameters;
	gPermanentArcLampGew : ArcLampGew_Parameters;
	gPermanentNirAdphos : NIRAdphos_Parameters;
	gPermanentCuringLed : ARRAY[0..2] OF CuringLed_Parameters_typ;
	gPermanentInkBox : InkboxParameters;
	gPermanentAnalogSensor : stThicknessAnalogPermanent;
END_VAR
```
